LIN {X 0,Y 312.686,Z 295.811,A -85,B 0,C 180,E1 -15649.642,E2 -15649.642} C_VEL
LIN {X 0,Y 312.798,Z 295.834,A -85,B 0,C 180,E1 -15652.253,E2 -15652.253} C_VEL
LIN {X 0,Y 312.699,Z 295.812,A -85,B 0,C 180,E1 -15654.843,E2 -15654.843} C_VEL
LIN {X 0,Y 312.984,Z 295.813,A -85,B 0,C 180,E1 -15658.714,E2 -15658.714} C_VEL
LIN {X 0,Y 312.982,Z 295.778,A -85,B 0,C 180,E1 -15661.287,E2 -15661.287} C_VEL
LIN {X 0,Y 312.841,Z 295.81,A -85,B 0,C 180,E1 -15666.484,E2 -15666.484} C_VEL
LIN {X 0,Y 312.753,Z 295.811,A -85,B 0,C 180,E1 -15669.051,E2 -15669.051} C_VEL
LIN {X 0,Y 312.634,Z 295.828,A -85,B 0,C 180,E1 -15672.992,E2 -15672.992} C_VEL
LIN {X 0,Y 312.615,Z 295.845,A -85,B 0,C 180,E1 -15675.652,E2 -15675.652} C_VEL
LIN {X 0,Y 312.536,Z 295.84,A -85,B 0,C 180,E1 -15679.714,E2 -15679.714} C_VEL
LIN {X 0,Y 312.516,Z 295.853,A -85,B 0,C 180,E1 -15682.775,E2 -15682.775} C_VEL
LIN {X 0,Y 312.491,Z 295.872,A -85,B 0,C 180,E1 -15684.987,E2 -15684.987} C_VEL
LIN {X 0,Y 313.356,Z 298.462,A -85,B 0,C 180,E1 -15685.341,E2 -15685.341} C_VEL
LIN {X 0,Y 315.346,Z 300.712,A -85,B 0,C 180,E1 -15685.986,E2 -15685.986} C_VEL
LIN {X 0,Y 316.693,Z 301.792,A -85,B 0,C 180,E1 -15686.394,E2 -15686.394} C_VEL
LIN {X 0,Y 318.598,Z 304.879,A -85,B 0,C 180,E1 -15687.019,E2 -15687.019} C_VEL
LIN {X 0,Y 320.808,Z 307.144,A -85,B 0,C 180,E1 -15687.673,E2 -15687.673} C_VEL
LIN {X 0,Y 323.371,Z 310.64,A -85,B 0,C 180,E1 -15688.44,E2 -15688.44} C_VEL
LIN {X 0,Y 324.737,Z 312.319,A -85,B 0,C 180,E1 -15688.831,E2 -15688.831} C_VEL
LIN {X 0,Y 328.562,Z 317.398,A -85,B 0,C 180,E1 -15689.896,E2 -15689.896} C_VEL
LIN {X 0,Y 334.896,Z 325.991,A -85,B 0,C 180,E1 -15691.559,E2 -15691.559} C_VEL
LIN {X 0,Y 343.13,Z 338.066,A -85,B 0,C 180,E1 -15693.575,E2 -15693.575} C_VEL
LIN {X 0,Y 348.752,Z 347.569,A -85,B 0,C 180,E1 -15694.885,E2 -15694.885} C_VEL
LIN {X 0,Y 355.328,Z 359.808,A -85,B 0,C 180,E1 -15696.353,E2 -15696.353} C_VEL
LIN {X 0,Y 348.994,Z 496.214,A -85,B 0,C 180,E1 -15699.224,E2 -15699.224} C_VEL
LIN {X 0,Y 347.586,Z 511.917,A -85,B 0,C 180,E1 -15699.738,E2 -15699.738} C_VEL
LIN {X 0,Y 345.628,Z 527.82,A -85,B 0,C 180,E1 -15700.466,E2 -15700.466} C_VEL
LIN {X 0,Y 343.213,Z 543.442,A -85,B 0,C 180,E1 -15701.412,E2 -15701.412} C_VEL
LIN {X 0,Y 340.307,Z 559.032,A -85,B 0,C 180,E1 -15702.615,E2 -15702.615} C_VEL
LIN {X 0,Y 337.092,Z 573.52,A -85,B 0,C 180,E1 -15704.004,E2 -15704.004} C_VEL
LIN {X 0,Y 333.707,Z 587.157,A -85,B 0,C 180,E1 -15705.595,E2 -15705.595} C_VEL
LIN {X 0,Y 330.15,Z 600.476,A -85,B 0,C 180,E1 -15707.478,E2 -15707.478} C_VEL
LIN {X 0,Y 326.807,Z 612.047,A -85,B 0,C 180,E1 -15709.427,E2 -15709.427} C_VEL
LIN {X 0,Y 323.531,Z 622.668,A -85,B 0,C 180,E1 -15711.558,E2 -15711.558} C_VEL
LIN {X 0,Y 320.715,Z 631.72,A -85,B 0,C 180,E1 -15713.724,E2 -15713.724} C_VEL
LIN {X 0,Y 317.842,Z 641.178,A -85,B 0,C 180,E1 -15716.441,E2 -15716.441} C_VEL
LIN {X 0,Y 315.491,Z 648.981,A -85,B 0,C 180,E1 -15719.179,E2 -15719.179} C_VEL
LIN {X 0,Y 313.706,Z 655.293,A -85,B 0,C 180,E1 -15721.935,E2 -15721.935} C_VEL
LIN {X 0,Y 312.36,Z 660.271,A -85,B 0,C 180,E1 -15724.691,E2 -15724.691} C_VEL
LIN {X 0,Y 311.406,Z 664.401,A -85,B 0,C 180,E1 -15727.717,E2 -15727.717} C_VEL
LIN {X 0,Y 310.878,Z 666.76,A -85,B 0,C 180,E1 -15730.178,E2 -15730.178} C_VEL
LIN {X 0,Y 310.594,Z 668.373,A -85,B 0,C 180,E1 -15732.893,E2 -15732.893} C_VEL
LIN {X 0,Y 310.522,Z 668.972,A -85,B 0,C 180,E1 -15735.584,E2 -15735.584} C_VEL
LIN {X 0,Y 310.539,Z 668.546,A -85,B 0,C 180,E1 -15738.247,E2 -15738.247} C_VEL
LIN {X 0,Y 310.551,Z 667.191,A -85,B 0,C 180,E1 -15740.885,E2 -15740.885} C_VEL
LIN {X 0,Y 310.957,Z 664.27,A -85,B 0,C 180,E1 -15743.971,E2 -15743.971} C_VEL
LIN {X 0,Y 311.31,Z 660.413,A -85,B 0,C 180,E1 -15746.764,E2 -15746.764} C_VEL
LIN {X 0,Y 311.935,Z 655.765,A -85,B 0,C 180,E1 -15749.354,E2 -15749.354} C_VEL
LIN {X 0,Y 313.296,Z 648.302,A -85,B 0,C 180,E1 -15752.571,E2 -15752.571} C_VEL
LIN {X 0,Y 314.909,Z 639.877,A -85,B 0,C 180,E1 -15755.443,E2 -15755.443} C_VEL
LIN {X 0,Y 316.998,Z 630.802,A -85,B 0,C 180,E1 -15757.965,E2 -15757.965} C_VEL
LIN {X 0,Y 319.443,Z 620.044,A -85,B 0,C 180,E1 -15760.457,E2 -15760.457} C_VEL
LIN {X 0,Y 321.871,Z 608.968,A -85,B 0,C 180,E1 -15762.612,E2 -15762.612} C_VEL
LIN {X 0,Y 324.394,Z 596.962,A -85,B 0,C 180,E1 -15764.587,E2 -15764.587} C_VEL
LIN {X 0,Y 327.032,Z 583.829,A -85,B 0,C 180,E1 -15766.383,E2 -15766.383} C_VEL
LIN {X 0,Y 329.507,Z 570.928,A -85,B 0,C 180,E1 -15767.854,E2 -15767.854} C_VEL
LIN {X 0,Y 332.094,Z 555.577,A -85,B 0,C 180,E1 -15769.309,E2 -15769.309} C_VEL
LIN {X 0,Y 334.275,Z 540.595,A -85,B 0,C 180,E1 -15770.459,E2 -15770.459} C_VEL
LIN {X 0,Y 335.936,Z 526.536,A -85,B 0,C 180,E1 -15771.315,E2 -15771.315} C_VEL
LIN {X 0,Y 337.496,Z 510.651,A -85,B 0,C 180,E1 -15772.054,E2 -15772.054} C_VEL
LIN {X 0,Y 338.691,Z 494.724,A -85,B 0,C 180,E1 -15772.574,E2 -15772.574} C_VEL
LIN {X 0,Y 341.33,Z 421.868,A -85,B 0,C 180,E1 -15774.13,E2 -15774.13} C_VEL
LIN {X 0,Y 340.959,Z 416.07,A -85,B 0,C 180,E1 -15774.315,E2 -15774.315} C_VEL
LIN {X 0,Y 336.956,Z 397.42,A -85,B 0,C 180,E1 -15775.237,E2 -15775.237} C_VEL
LIN {X 0,Y 336.559,Z 391.625,A -85,B 0,C 180,E1 -15775.431,E2 -15775.431} C_VEL
LIN {X 0,Y 338.038,Z 354.66,A -85,B 0,C 180,E1 -15776.204,E2 -15776.204} C_VEL
LIN {X 0,Y 328.733,Z 335.509,A -85,B 0,C 180,E1 -15777.866,E2 -15777.866} C_VEL
LIN {X 0,Y 318.795,Z 318.498,A -85,B 0,C 180,E1 -15779.685,E2 -15779.685} C_VEL
LIN {X 0,Y 309.969,Z 304.705,A -85,B 0,C 180,E1 -15781.395,E2 -15781.395} C_VEL
LIN {X 0,Y 307.637,Z 301.06,A -85,B 0,C 180,E1 -15781.869,E2 -15781.869} C_VEL
LIN {X 0,Y 305.928,Z 298.586,A -85,B 0,C 180,E1 -15782.217,E2 -15782.217} C_VEL
LIN {X 0,Y 305.465,Z 296.743,A -85,B 0,C 180,E1 -15782.352,E2 -15782.352} C_VEL
LIN {X 0,Y 305.464,Z 296.749,A -85,B 0,C 180,E1 -15786.363,E2 -15786.363} C_VEL
LIN {X 0,Y 305.412,Z 296.756,A -85,B 0,C 180,E1 -15790.115,E2 -15790.115} C_VEL
LIN {X 0,Y 305.422,Z 296.75,A -85,B 0,C 180,E1 -15793.656,E2 -15793.656} C_VEL
LIN {X 0,Y 305.436,Z 296.74,A -85,B 0,C 180,E1 -15797.418,E2 -15797.418} C_VEL
LIN {X 0,Y 305.449,Z 296.709,A -85,B 0,C 180,E1 -15801.593,E2 -15801.593} C_VEL
LIN {X 0,Y 305.462,Z 296.701,A -85,B 0,C 180,E1 -15804.886,E2 -15804.886} C_VEL
LIN {X 0,Y 305.443,Z 296.75,A -85,B 0,C 180,E1 -15808.358,E2 -15808.358} C_VEL
LIN {X 0,Y 305.455,Z 296.731,A -85,B 0,C 180,E1 -15811.106,E2 -15811.106} C_VEL
LIN {X 0,Y 305.499,Z 296.741,A -85,B 0,C 180,E1 -15814.081,E2 -15814.081} C_VEL
LIN {X 0,Y 305.475,Z 296.73,A -85,B 0,C 180,E1 -15816.975,E2 -15816.975} C_VEL
LIN {X 0,Y 305.544,Z 296.724,A -85,B 0,C 180,E1 -15821.214,E2 -15821.214} C_VEL
LIN {X 0,Y 305.628,Z 296.729,A -85,B 0,C 180,E1 -15825.347,E2 -15825.347} C_VEL
LIN {X 0,Y 305.636,Z 296.713,A -85,B 0,C 180,E1 -15829.399,E2 -15829.399} C_VEL
LIN {X 0,Y 305.772,Z 296.706,A -85,B 0,C 180,E1 -15832.073,E2 -15832.073} C_VEL
LIN {X 0,Y 305.675,Z 296.702,A -85,B 0,C 180,E1 -15834.722,E2 -15834.722} C_VEL
LIN {X 0,Y 305.954,Z 296.681,A -85,B 0,C 180,E1 -15838.683,E2 -15838.683} C_VEL
LIN {X 0,Y 305.954,Z 296.669,A -85,B 0,C 180,E1 -15841.316,E2 -15841.316} C_VEL
LIN {X 0,Y 305.679,Z 296.707,A -85,B 0,C 180,E1 -15845.276,E2 -15845.276} C_VEL
LIN {X 0,Y 305.799,Z 296.68,A -85,B 0,C 180,E1 -15847.925,E2 -15847.925} C_VEL
LIN {X 0,Y 305.603,Z 296.725,A -85,B 0,C 180,E1 -15851.944,E2 -15851.944} C_VEL
LIN {X 0,Y 305.608,Z 296.729,A -85,B 0,C 180,E1 -15855.014,E2 -15855.014} C_VEL
LIN {X 0,Y 305.56,Z 296.734,A -85,B 0,C 180,E1 -15859.436,E2 -15859.436} C_VEL
LIN {X 0,Y 305.49,Z 296.744,A -85,B 0,C 180,E1 -15863.041,E2 -15863.041} C_VEL
LIN {X 0,Y 305.53,Z 296.741,A -85,B 0,C 180,E1 -15866.22,E2 -15866.22} C_VEL
LIN {X 0,Y 305.487,Z 296.746,A -85,B 0,C 180,E1 -15869.047,E2 -15869.047} C_VEL
LIN {X 0,Y 305.44,Z 296.752,A -85,B 0,C 180,E1 -15871.952,E2 -15871.952} C_VEL
LIN {X 0,Y 305.461,Z 296.744,A -85,B 0,C 180,E1 -15875.113,E2 -15875.113} C_VEL
LIN {X 0,Y 305.465,Z 296.748,A -85,B 0,C 180,E1 -15878.533,E2 -15878.533} C_VEL
LIN {X 0,Y 305.457,Z 296.753,A -85,B 0,C 180,E1 -15882.586,E2 -15882.586} C_VEL
LIN {X 0,Y 305.427,Z 296.81,A -85,B 0,C 180,E1 -15883.063,E2 -15883.063} C_VEL
LIN {X 0,Y 308.169,Z 304.268,A -85,B 0,C 180,E1 -15884.928,E2 -15884.928} C_VEL
LIN {X 0,Y 316.716,Z 319.019,A -85,B 0,C 180,E1 -15886.646,E2 -15886.646} C_VEL
LIN {X 0,Y 323.706,Z 332.142,A -85,B 0,C 180,E1 -15887.992,E2 -15887.992} C_VEL
LIN {X 0,Y 332.604,Z 350.491,A -85,B 0,C 180,E1 -15889.641,E2 -15889.641} C_VEL
LIN {X 0,Y 337.927,Z 362.483,A -85,B 0,C 180,E1 -15890.598,E2 -15890.598} C_VEL
LIN {X 0,Y 332.319,Z 511.428,A -85,B 0,C 180,E1 -15893.784,E2 -15893.784} C_VEL
LIN {X 0,Y 331.012,Z 527.703,A -85,B 0,C 180,E1 -15894.323,E2 -15894.323} C_VEL
LIN {X 0,Y 329.18,Z 543.894,A -85,B 0,C 180,E1 -15895.079,E2 -15895.079} C_VEL
LIN {X 0,Y 327.159,Z 559.351,A -85,B 0,C 180,E1 -15896.046,E2 -15896.046} C_VEL
LIN {X 0,Y 324.616,Z 574.513,A -85,B 0,C 180,E1 -15897.231,E2 -15897.231} C_VEL
LIN {X 0,Y 322.08,Z 588.525,A -85,B 0,C 180,E1 -15898.603,E2 -15898.603} C_VEL
LIN {X 0,Y 319.117,Z 602.903,A -85,B 0,C 180,E1 -15900.296,E2 -15900.296} C_VEL
LIN {X 0,Y 316.291,Z 616.145,A -85,B 0,C 180,E1 -15902.185,E2 -15902.185} C_VEL
LIN {X 0,Y 313.742,Z 627.491,A -85,B 0,C 180,E1 -15904.1,E2 -15904.1} C_VEL
LIN {X 0,Y 311.182,Z 638.736,A -85,B 0,C 180,E1 -15906.367,E2 -15906.367} C_VEL
LIN {X 0,Y 309.055,Z 648.356,A -85,B 0,C 180,E1 -15908.664,E2 -15908.664} C_VEL
LIN {X 0,Y 307.152,Z 657.693,A -85,B 0,C 180,E1 -15911.317,E2 -15911.317} C_VEL
LIN {X 0,Y 305.648,Z 665.471,A -85,B 0,C 180,E1 -15913.983,E2 -15913.983} C_VEL
LIN {X 0,Y 304.665,Z 671.817,A -85,B 0,C 180,E1 -15916.663,E2 -15916.663} C_VEL
LIN {X 0,Y 303.958,Z 676.988,A -85,B 0,C 180,E1 -15919.341,E2 -15919.341} C_VEL
LIN {X 0,Y 303.682,Z 680.998,A -85,B 0,C 180,E1 -15922.019,E2 -15922.019} C_VEL
LIN {X 0,Y 303.614,Z 683.933,A -85,B 0,C 180,E1 -15924.687,E2 -15924.687} C_VEL
LIN {X 0,Y 303.601,Z 685.852,A -85,B 0,C 180,E1 -15927.347,E2 -15927.347} C_VEL
LIN {X 0,Y 303.602,Z 686.754,A -85,B 0,C 180,E1 -15930,E2 -15930} C_VEL
LIN {X 0,Y 303.592,Z 686.701,A -85,B 0,C 180,E1 -15932.654,E2 -15932.654} C_VEL
LIN {X 0,Y 303.621,Z 685.522,A -85,B 0,C 180,E1 -15935.545,E2 -15935.545} C_VEL
LIN {X 0,Y 303.688,Z 683.676,A -85,B 0,C 180,E1 -15937.982,E2 -15937.982} C_VEL
LIN {X 0,Y 304.027,Z 680.69,A -85,B 0,C 180,E1 -15940.657,E2 -15940.657} C_VEL
LIN {X 0,Y 304.827,Z 676.704,A -85,B 0,C 180,E1 -15943.33,E2 -15943.33} C_VEL
LIN {X 0,Y 305.923,Z 671.604,A -85,B 0,C 180,E1 -15946.003,E2 -15946.003} C_VEL
LIN {X 0,Y 307.626,Z 665.419,A -85,B 0,C 180,E1 -15948.654,E2 -15948.654} C_VEL
LIN {X 0,Y 309.772,Z 657.865,A -85,B 0,C 180,E1 -15951.285,E2 -15951.285} C_VEL
LIN {X 0,Y 312.559,Z 648.91,A -85,B 0,C 180,E1 -15953.875,E2 -15953.875} C_VEL
LIN {X 0,Y 315.874,Z 638.315,A -85,B 0,C 180,E1 -15956.423,E2 -15956.423} C_VEL
LIN {X 0,Y 319.215,Z 627.6,A -85,B 0,C 180,E1 -15958.575,E2 -15958.575} C_VEL
LIN {X 0,Y 322.531,Z 616.502,A -85,B 0,C 180,E1 -15960.439,E2 -15960.439} C_VEL
LIN {X 0,Y 325.907,Z 605.036,A -85,B 0,C 180,E1 -15962.075,E2 -15962.075} C_VEL
LIN {X 0,Y 329.415,Z 591.636,A -85,B 0,C 180,E1 -15963.691,E2 -15963.691} C_VEL
LIN {X 0,Y 332.99,Z 577.061,A -85,B 0,C 180,E1 -15965.109,E2 -15965.109} C_VEL
LIN {X 0,Y 335.929,Z 563.101,A -85,B 0,C 180,E1 -15966.23,E2 -15966.23} C_VEL
LIN {X 0,Y 338.617,Z 548.294,A -85,B 0,C 180,E1 -15967.192,E2 -15967.192} C_VEL
LIN {X 0,Y 341.085,Z 531.799,A -85,B 0,C 180,E1 -15967.994,E2 -15967.994} C_VEL
LIN {X 0,Y 342.849,Z 515.977,A -85,B 0,C 180,E1 -15968.542,E2 -15968.542} C_VEL
LIN {X 0,Y 344.097,Z 495.089,A -85,B 0,C 180,E1 -15969.047,E2 -15969.047} C_VEL
LIN {X 0,Y 349.94,Z 369.642,A -85,B 0,C 180,E1 -15971.705,E2 -15971.705} C_VEL
LIN {X 0,Y 342.001,Z 354.097,A -85,B 0,C 180,E1 -15973.584,E2 -15973.584} C_VEL
LIN {X 0,Y 334.526,Z 340.991,A -85,B 0,C 180,E1 -15975.465,E2 -15975.465} C_VEL
LIN {X 0,Y 327.373,Z 329.638,A -85,B 0,C 180,E1 -15977.385,E2 -15977.385} C_VEL
LIN {X 0,Y 320.557,Z 319.554,A -85,B 0,C 180,E1 -15979.362,E2 -15979.362} C_VEL
LIN {X 0,Y 316.114,Z 313.396,A -85,B 0,C 180,E1 -15980.742,E2 -15980.742} C_VEL
LIN {X 0,Y 309.814,Z 305.018,A -85,B 0,C 180,E1 -15982.846,E2 -15982.846} C_VEL
LIN {X 0,Y 307.631,Z 301.915,A -85,B 0,C 180,E1 -15983.669,E2 -15983.669} C_VEL
LIN {X 0,Y 305.507,Z 297.046,A -85,B 0,C 180,E1 -15985.756,E2 -15985.756} C_VEL
LIN {X 0,Y 305.464,Z 296.728,A -85,B 0,C 180,E1 -15985.922,E2 -15985.922} C_VEL
LIN {X 0,Y 305.459,Z 296.748,A -85,B 0,C 180,E1 -15989.591,E2 -15989.591} C_VEL
LIN {X 0,Y 305.518,Z 296.713,A -85,B 0,C 180,E1 -15992.609,E2 -15992.609} C_VEL
LIN {X 0,Y 305.505,Z 296.728,A -85,B 0,C 180,E1 -15995.539,E2 -15995.539} C_VEL
LIN {X 0,Y 305.513,Z 296.741,A -85,B 0,C 180,E1 -15999.815,E2 -15999.815} C_VEL
LIN {X 0,Y 305.575,Z 296.7,A -85,B 0,C 180,E1 -16002.604,E2 -16002.604} C_VEL
LIN {X 0,Y 305.65,Z 296.715,A -85,B 0,C 180,E1 -16005.35,E2 -16005.35} C_VEL
LIN {X 0,Y 305.625,Z 296.689,A -85,B 0,C 180,E1 -16009.4,E2 -16009.4} C_VEL
LIN {X 0,Y 305.748,Z 296.711,A -85,B 0,C 180,E1 -16012.073,E2 -16012.073} C_VEL
LIN {X 0,Y 305.668,Z 296.688,A -85,B 0,C 180,E1 -16014.724,E2 -16014.724} C_VEL
LIN {X 0,Y 305.951,Z 296.689,A -85,B 0,C 180,E1 -16018.684,E2 -16018.684} C_VEL
LIN {X 0,Y 305.949,Z 296.653,A -85,B 0,C 180,E1 -16021.317,E2 -16021.317} C_VEL
LIN {X 0,Y 305.789,Z 296.685,A -85,B 0,C 180,E1 -16026.6,E2 -16026.6} C_VEL
LIN {X 0,Y 305.696,Z 296.692,A -85,B 0,C 180,E1 -16029.262,E2 -16029.262} C_VEL
LIN {X 0,Y 305.587,Z 296.702,A -85,B 0,C 180,E1 -16033.297,E2 -16033.297} C_VEL
LIN {X 0,Y 305.543,Z 296.733,A -85,B 0,C 180,E1 -16036.024,E2 -16036.024} C_VEL
LIN {X 0,Y 305.482,Z 296.723,A -85,B 0,C 180,E1 -16040.188,E2 -16040.188} C_VEL
LIN {X 0,Y 305.47,Z 296.729,A -85,B 0,C 180,E1 -16042.879,E2 -16042.879} C_VEL
LIN {X 0,Y 306.272,Z 299.3,A -85,B 0,C 180,E1 -16043.267,E2 -16043.267} C_VEL
LIN {X 0,Y 308.202,Z 301.528,A -85,B 0,C 180,E1 -16043.966,E2 -16043.966} C_VEL
LIN {X 0,Y 309.717,Z 302.518,A -85,B 0,C 180,E1 -16044.465,E2 -16044.465} C_VEL
LIN {X 0,Y 311.507,Z 305.592,A -85,B 0,C 180,E1 -16045.116,E2 -16045.116} C_VEL
LIN {X 0,Y 313.981,Z 308.059,A -85,B 0,C 180,E1 -16045.912,E2 -16045.912} C_VEL
LIN {X 0,Y 316.359,Z 311.432,A -85,B 0,C 180,E1 -16046.691,E2 -16046.691} C_VEL
LIN {X 0,Y 317.908,Z 313.042,A -85,B 0,C 180,E1 -16047.161,E2 -16047.161} C_VEL
LIN {X 0,Y 320.945,Z 317.023,A -85,B 0,C 180,E1 -16048.085,E2 -16048.085} C_VEL
LIN {X 0,Y 325.541,Z 323.245,A -85,B 0,C 180,E1 -16049.417,E2 -16049.417} C_VEL
LIN {X 0,Y 332.025,Z 332.219,A -85,B 0,C 180,E1 -16051.166,E2 -16051.166} C_VEL
LIN {X 0,Y 339.376,Z 343.096,A -85,B 0,C 180,E1 -16053.018,E2 -16053.018} C_VEL
LIN {X 0,Y 344.768,Z 352.352,A -85,B 0,C 180,E1 -16054.317,E2 -16054.317} C_VEL
LIN {X 0,Y 350.248,Z 362.537,A -85,B 0,C 180,E1 -16055.586,E2 -16055.586} C_VEL
LIN {X 0,Y 343.759,Z 496.864,A -85,B 0,C 180,E1 -16058.442,E2 -16058.442} C_VEL
LIN {X 0,Y 342.305,Z 512.312,A -85,B 0,C 180,E1 -16058.956,E2 -16058.956} C_VEL
LIN {X 0,Y 340.414,Z 527.383,A -85,B 0,C 180,E1 -16059.651,E2 -16059.651} C_VEL
LIN {X 0,Y 337.874,Z 543.192,A -85,B 0,C 180,E1 -16060.604,E2 -16060.604} C_VEL
LIN {X 0,Y 334.822,Z 558.968,A -85,B 0,C 180,E1 -16061.828,E2 -16061.828} C_VEL
LIN {X 0,Y 331.523,Z 573.382,A -85,B 0,C 180,E1 -16063.22,E2 -16063.22} C_VEL
LIN {X 0,Y 328.055,Z 586.826,A -85,B 0,C 180,E1 -16064.794,E2 -16064.794} C_VEL
LIN {X 0,Y 324.267,Z 600.442,A -85,B 0,C 180,E1 -16066.731,E2 -16066.731} C_VEL
LIN {X 0,Y 320.961,Z 611.512,A -85,B 0,C 180,E1 -16068.605,E2 -16068.605} C_VEL
LIN {X 0,Y 317.441,Z 622.344,A -85,B 0,C 180,E1 -16070.796,E2 -16070.796} C_VEL
LIN {X 0,Y 314.234,Z 632.134,A -85,B 0,C 180,E1 -16073.169,E2 -16073.169} C_VEL
LIN {X 0,Y 311.495,Z 640.718,A -85,B 0,C 180,E1 -16075.663,E2 -16075.663} C_VEL
LIN {X 0,Y 308.963,Z 648.648,A -85,B 0,C 180,E1 -16078.454,E2 -16078.454} C_VEL
LIN {X 0,Y 307.008,Z 655.035,A -85,B 0,C 180,E1 -16081.267,E2 -16081.267} C_VEL
LIN {X 0,Y 305.53,Z 660.135,A -85,B 0,C 180,E1 -16084.084,E2 -16084.084} C_VEL
LIN {X 0,Y 304.548,Z 664.073,A -85,B 0,C 180,E1 -16086.902,E2 -16086.902} C_VEL
LIN {X 0,Y 303.888,Z 666.788,A -85,B 0,C 180,E1 -16089.702,E2 -16089.702} C_VEL
LIN {X 0,Y 303.537,Z 668.506,A -85,B 0,C 180,E1 -16092.482,E2 -16092.482} C_VEL
LIN {X 0,Y 303.42,Z 669.157,A -85,B 0,C 180,E1 -16095.239,E2 -16095.239} C_VEL
LIN {X 0,Y 303.433,Z 668.835,A -85,B 0,C 180,E1 -16097.968,E2 -16097.968} C_VEL
LIN {X 0,Y 303.445,Z 667.529,A -85,B 0,C 180,E1 -16100.67,E2 -16100.67} C_VEL
LIN {X 0,Y 303.883,Z 664.542,A -85,B 0,C 180,E1 -16103.983,E2 -16103.983} C_VEL
LIN {X 0,Y 304.194,Z 660.962,A -85,B 0,C 180,E1 -16106.689,E2 -16106.689} C_VEL
LIN {X 0,Y 304.852,Z 656.366,A -85,B 0,C 180,E1 -16109.339,E2 -16109.339} C_VEL
LIN {X 0,Y 305.899,Z 650.613,A -85,B 0,C 180,E1 -16111.975,E2 -16111.975} C_VEL
LIN {X 0,Y 307.221,Z 643.701,A -85,B 0,C 180,E1 -16114.592,E2 -16114.592} C_VEL
LIN {X 0,Y 309.122,Z 635.333,A -85,B 0,C 180,E1 -16117.183,E2 -16117.183} C_VEL
LIN {X 0,Y 311.52,Z 625.363,A -85,B 0,C 180,E1 -16119.741,E2 -16119.741} C_VEL
LIN {X 0,Y 313.901,Z 615.131,A -85,B 0,C 180,E1 -16121.952,E2 -16121.952} C_VEL
LIN {X 0,Y 316.599,Z 603.168,A -85,B 0,C 180,E1 -16124.133,E2 -16124.133} C_VEL
LIN {X 0,Y 319.2,Z 591.124,A -85,B 0,C 180,E1 -16125.975,E2 -16125.975} C_VEL
LIN {X 0,Y 321.797,Z 578.151,A -85,B 0,C 180,E1 -16127.639,E2 -16127.639} C_VEL
LIN {X 0,Y 324.447,Z 564.219,A -85,B 0,C 180,E1 -16129.125,E2 -16129.125} C_VEL
LIN {X 0,Y 326.846,Z 549.19,A -85,B 0,C 180,E1 -16130.451,E2 -16130.451} C_VEL
LIN {X 0,Y 328.957,Z 533.645,A -85,B 0,C 180,E1 -16131.543,E2 -16131.543} C_VEL
LIN {X 0,Y 330.945,Z 516.706,A -85,B 0,C 180,E1 -16132.432,E2 -16132.432} C_VEL
LIN {X 0,Y 332.211,Z 501.941,A -85,B 0,C 180,E1 -16132.999,E2 -16132.999} C_VEL
LIN {X 0,Y 333.161,Z 484.122,A -85,B 0,C 180,E1 -16133.463,E2 -16133.463} C_VEL
LIN {X 0,Y 336.559,Z 391.625,A -85,B 0,C 180,E1 -16135.431,E2 -16135.431} C_VEL
LIN {X 0,Y 336.151,Z 385.828,A -85,B 0,C 180,E1 -16135.627,E2 -16135.627} C_VEL
LIN {X 0,Y 332.238,Z 367.184,A -85,B 0,C 180,E1 -16136.581,E2 -16136.581} C_VEL
LIN {X 0,Y 331.992,Z 361.383,A -85,B 0,C 180,E1 -16136.764,E2 -16136.764} C_VEL
LIN {X 0,Y 332.117,Z 356.706,A -85,B 0,C 180,E1 -16136.872,E2 -16136.872} C_VEL
LIN {X 0,Y 323.631,Z 339.316,A -85,B 0,C 180,E1 -16138.434,E2 -16138.434} C_VEL
LIN {X 0,Y 314.098,Z 322.876,A -85,B 0,C 180,E1 -16140.239,E2 -16140.239} C_VEL
LIN {X 0,Y 305.424,Z 309.288,A -85,B 0,C 180,E1 -16141.97,E2 -16141.97} C_VEL
LIN {X 0,Y 303.104,Z 305.75,A -85,B 0,C 180,E1 -16142.455,E2 -16142.455} C_VEL
LIN {X 0,Y 300.673,Z 301.985,A -85,B 0,C 180,E1 -16142.976,E2 -16142.976} C_VEL
LIN {X 0,Y 298.963,Z 299.557,A -85,B 0,C 180,E1 -16143.344,E2 -16143.344} C_VEL
LIN {X 0,Y 298.436,Z 297.626,A -85,B 0,C 180,E1 -16143.515,E2 -16143.515} C_VEL
LIN {X 0,Y 298.389,Z 297.62,A -85,B 0,C 180,E1 -16147.762,E2 -16147.762} C_VEL
LIN {X 0,Y 298.349,Z 297.625,A -85,B 0,C 180,E1 -16151.267,E2 -16151.267} C_VEL
LIN {X 0,Y 298.357,Z 297.629,A -85,B 0,C 180,E1 -16155.034,E2 -16155.034} C_VEL
LIN {X 0,Y 298.349,Z 297.634,A -85,B 0,C 180,E1 -16158.921,E2 -16158.921} C_VEL
LIN {X 0,Y 298.427,Z 297.564,A -85,B 0,C 180,E1 -16163.197,E2 -16163.197} C_VEL
LIN {X 0,Y 298.394,Z 297.623,A -85,B 0,C 180,E1 -16167.199,E2 -16167.199} C_VEL
LIN {X 0,Y 298.366,Z 297.613,A -85,B 0,C 180,E1 -16170.637,E2 -16170.637} C_VEL
LIN {X 0,Y 298.439,Z 297.615,A -85,B 0,C 180,E1 -16174.919,E2 -16174.919} C_VEL
LIN {X 0,Y 298.404,Z 297.619,A -85,B 0,C 180,E1 -16177.862,E2 -16177.862} C_VEL
LIN {X 0,Y 298.505,Z 297.606,A -85,B 0,C 180,E1 -16180.754,E2 -16180.754} C_VEL
LIN {X 0,Y 298.587,Z 297.604,A -85,B 0,C 180,E1 -16184.994,E2 -16184.994} C_VEL
LIN {X 0,Y 298.592,Z 297.588,A -85,B 0,C 180,E1 -16189.146,E2 -16189.146} C_VEL
LIN {X 0,Y 298.718,Z 297.585,A -85,B 0,C 180,E1 -16191.884,E2 -16191.884} C_VEL
LIN {X 0,Y 298.645,Z 297.576,A -85,B 0,C 180,E1 -16194.598,E2 -16194.598} C_VEL
LIN {X 0,Y 298.92,Z 297.557,A -85,B 0,C 180,E1 -16198.652,E2 -16198.652} C_VEL
LIN {X 0,Y 298.921,Z 297.545,A -85,B 0,C 180,E1 -16201.346,E2 -16201.346} C_VEL
LIN {X 0,Y 298.65,Z 297.58,A -85,B 0,C 180,E1 -16205.401,E2 -16205.401} C_VEL
LIN {X 0,Y 298.743,Z 297.56,A -85,B 0,C 180,E1 -16208.114,E2 -16208.114} C_VEL
LIN {X 0,Y 298.553,Z 297.602,A -85,B 0,C 180,E1 -16212.231,E2 -16212.231} C_VEL
LIN {X 0,Y 298.548,Z 297.607,A -85,B 0,C 180,E1 -16215.168,E2 -16215.168} C_VEL
LIN {X 0,Y 298.52,Z 297.61,A -85,B 0,C 180,E1 -16219.244,E2 -16219.244} C_VEL
LIN {X 0,Y 298.457,Z 297.624,A -85,B 0,C 180,E1 -16223.597,E2 -16223.597} C_VEL
LIN {X 0,Y 298.485,Z 297.62,A -85,B 0,C 180,E1 -16226.574,E2 -16226.574} C_VEL
LIN {X 0,Y 298.415,Z 297.628,A -85,B 0,C 180,E1 -16229.641,E2 -16229.641} C_VEL
LIN {X 0,Y 298.393,Z 297.627,A -85,B 0,C 180,E1 -16232.8,E2 -16232.8} C_VEL
LIN {X 0,Y 298.445,Z 297.605,A -85,B 0,C 180,E1 -16236.807,E2 -16236.807} C_VEL
LIN {X 0,Y 298.407,Z 297.624,A -85,B 0,C 180,E1 -16239.486,E2 -16239.486} C_VEL
LIN {X 0,Y 298.431,Z 297.817,A -85,B 0,C 180,E1 -16242.1,E2 -16242.1} C_VEL
LIN {X 0,Y 300.758,Z 303.975,A -85,B 0,C 180,E1 -16243.716,E2 -16243.716} C_VEL
LIN {X 0,Y 310.516,Z 320.667,A -85,B 0,C 180,E1 -16245.78,E2 -16245.78} C_VEL
LIN {X 0,Y 318.198,Z 335.006,A -85,B 0,C 180,E1 -16247.313,E2 -16247.313} C_VEL
LIN {X 0,Y 327.233,Z 353.65,A -85,B 0,C 180,E1 -16249.044,E2 -16249.044} C_VEL
LIN {X 0,Y 332.038,Z 364.587,A -85,B 0,C 180,E1 -16249.942,E2 -16249.942} C_VEL
LIN {X 0,Y 326.268,Z 512.099,A -85,B 0,C 180,E1 -16253.147,E2 -16253.147} C_VEL
LIN {X 0,Y 324.827,Z 528.962,A -85,B 0,C 180,E1 -16253.729,E2 -16253.729} C_VEL
LIN {X 0,Y 322.946,Z 544.74,A -85,B 0,C 180,E1 -16254.495,E2 -16254.495} C_VEL
LIN {X 0,Y 320.713,Z 560.972,A -85,B 0,C 180,E1 -16255.553,E2 -16255.553} C_VEL
LIN {X 0,Y 317.909,Z 576.606,A -85,B 0,C 180,E1 -16256.826,E2 -16256.826} C_VEL
LIN {X 0,Y 315.073,Z 591.772,A -85,B 0,C 180,E1 -16258.386,E2 -16258.386} C_VEL
LIN {X 0,Y 312.083,Z 605.599,A -85,B 0,C 180,E1 -16260.116,E2 -16260.116} C_VEL
LIN {X 0,Y 309.424,Z 617.357,A -85,B 0,C 180,E1 -16261.882,E2 -16261.882} C_VEL
LIN {X 0,Y 306.841,Z 628.501,A -85,B 0,C 180,E1 -16263.838,E2 -16263.838} C_VEL
LIN {X 0,Y 304.201,Z 639.609,A -85,B 0,C 180,E1 -16266.153,E2 -16266.153} C_VEL
LIN {X 0,Y 301.939,Z 649.407,A -85,B 0,C 180,E1 -16268.597,E2 -16268.597} C_VEL
LIN {X 0,Y 300.067,Z 658.219,A -85,B 0,C 180,E1 -16271.214,E2 -16271.214} C_VEL
LIN {X 0,Y 298.712,Z 664.999,A -85,B 0,C 180,E1 -16273.601,E2 -16273.601} C_VEL
LIN {X 0,Y 297.676,Z 671.406,A -85,B 0,C 180,E1 -16276.344,E2 -16276.344} C_VEL
LIN {X 0,Y 296.908,Z 676.63,A -85,B 0,C 180,E1 -16279.084,E2 -16279.084} C_VEL
LIN {X 0,Y 296.614,Z 680.667,A -85,B 0,C 180,E1 -16281.827,E2 -16281.827} C_VEL
LIN {X 0,Y 296.548,Z 683.65,A -85,B 0,C 180,E1 -16284.56,E2 -16284.56} C_VEL
LIN {X 0,Y 296.526,Z 685.591,A -85,B 0,C 180,E1 -16287.283,E2 -16287.283} C_VEL
LIN {X 0,Y 296.517,Z 686.535,A -85,B 0,C 180,E1 -16290,E2 -16290} C_VEL
LIN {X 0,Y 296.516,Z 686.505,A -85,B 0,C 180,E1 -16292.717,E2 -16292.717} C_VEL
LIN {X 0,Y 296.508,Z 685.511,A -85,B 0,C 180,E1 -16295.441,E2 -16295.441} C_VEL
LIN {X 0,Y 296.621,Z 683.546,A -85,B 0,C 180,E1 -16298.173,E2 -16298.173} C_VEL
LIN {X 0,Y 296.986,Z 680.606,A -85,B 0,C 180,E1 -16300.913,E2 -16300.913} C_VEL
LIN {X 0,Y 297.848,Z 676.644,A -85,B 0,C 180,E1 -16303.648,E2 -16303.648} C_VEL
LIN {X 0,Y 299.012,Z 671.596,A -85,B 0,C 180,E1 -16306.383,E2 -16306.383} C_VEL
LIN {X 0,Y 300.828,Z 665.443,A -85,B 0,C 180,E1 -16309.091,E2 -16309.091} C_VEL
LIN {X 0,Y 303.468,Z 656.884,A -85,B 0,C 180,E1 -16312.128,E2 -16312.128} C_VEL
LIN {X 0,Y 306.416,Z 647.843,A -85,B 0,C 180,E1 -16314.745,E2 -16314.745} C_VEL
LIN {X 0,Y 309.971,Z 637.143,A -85,B 0,C 180,E1 -16317.314,E2 -16317.314} C_VEL
LIN {X 0,Y 313.567,Z 626.004,A -85,B 0,C 180,E1 -16319.544,E2 -16319.544} C_VEL
LIN {X 0,Y 317.591,Z 612.979,A -85,B 0,C 180,E1 -16321.707,E2 -16321.707} C_VEL
LIN {X 0,Y 321.838,Z 598.764,A -85,B 0,C 180,E1 -16323.618,E2 -16323.618} C_VEL
LIN {X 0,Y 325.389,Z 585.329,A -85,B 0,C 180,E1 -16325.105,E2 -16325.105} C_VEL
LIN {X 0,Y 328.768,Z 571.267,A -85,B 0,C 180,E1 -16326.385,E2 -16326.385} C_VEL
LIN {X 0,Y 331.9,Z 556.173,A -85,B 0,C 180,E1 -16327.502,E2 -16327.502} C_VEL
LIN {X 0,Y 334.298,Z 542.026,A -85,B 0,C 180,E1 -16328.33,E2 -16328.33} C_VEL
LIN {X 0,Y 336.603,Z 525.612,A -85,B 0,C 180,E1 -16329.045,E2 -16329.045} C_VEL
LIN {X 0,Y 338.277,Z 508.622,A -85,B 0,C 180,E1 -16329.557,E2 -16329.557} C_VEL
LIN {X 0,Y 344.913,Z 372.333,A -85,B 0,C 180,E1 -16332.496,E2 -16332.496} C_VEL
LIN {X 0,Y 337.445,Z 357.745,A -85,B 0,C 180,E1 -16334.335,E2 -16334.335} C_VEL
LIN {X 0,Y 331.112,Z 346.439,A -85,B 0,C 180,E1 -16335.992,E2 -16335.992} C_VEL
LIN {X 0,Y 324.191,Z 335.26,A -85,B 0,C 180,E1 -16337.908,E2 -16337.908} C_VEL
LIN {X 0,Y 317.066,Z 324.592,A -85,B 0,C 180,E1 -16340.051,E2 -16340.051} C_VEL
LIN {X 0,Y 313.067,Z 318.986,A -85,B 0,C 180,E1 -16341.337,E2 -16341.337} C_VEL
LIN {X 0,Y 307.372,Z 311.224,A -85,B 0,C 180,E1 -16343.302,E2 -16343.302} C_VEL
LIN {X 0,Y 303.646,Z 306.318,A -85,B 0,C 180,E1 -16344.697,E2 -16344.697} C_VEL
LIN {X 0,Y 301.002,Z 302.932,A -85,B 0,C 180,E1 -16345.741,E2 -16345.741} C_VEL
LIN {X 0,Y 300.205,Z 301.46,A -85,B 0,C 180,E1 -16346.12,E2 -16346.12} C_VEL
LIN {X 0,Y 298.84,Z 299.363,A -85,B 0,C 180,E1 -16347.256,E2 -16347.256} C_VEL
LIN {X 0,Y 298.397,Z 297.608,A -85,B 0,C 180,E1 -16348.103,E2 -16348.103} C_VEL
LIN {X 0,Y 298.459,Z 297.589,A -85,B 0,C 180,E1 -16351.905,E2 -16351.905} C_VEL
LIN {X 0,Y 298.484,Z 297.615,A -85,B 0,C 180,E1 -16354.925,E2 -16354.925} C_VEL
LIN {X 0,Y 298.441,Z 297.61,A -85,B 0,C 180,E1 -16359.315,E2 -16359.315} C_VEL
LIN {X 0,Y 298.538,Z 297.58,A -85,B 0,C 180,E1 -16362.18,E2 -16362.18} C_VEL
LIN {X 0,Y 298.594,Z 297.585,A -85,B 0,C 180,E1 -16364.996,E2 -16364.996} C_VEL
LIN {X 0,Y 298.584,Z 297.566,A -85,B 0,C 180,E1 -16369.147,E2 -16369.147} C_VEL
LIN {X 0,Y 298.7,Z 297.586,A -85,B 0,C 180,E1 -16371.885,E2 -16371.885} C_VEL
LIN {X 0,Y 298.637,Z 297.565,A -85,B 0,C 180,E1 -16374.599,E2 -16374.599} C_VEL
LIN {X 0,Y 298.918,Z 297.564,A -85,B 0,C 180,E1 -16378.653,E2 -16378.653} C_VEL
LIN {X 0,Y 298.915,Z 297.527,A -85,B 0,C 180,E1 -16381.348,E2 -16381.348} C_VEL
LIN {X 0,Y 298.738,Z 297.56,A -85,B 0,C 180,E1 -16386.756,E2 -16386.756} C_VEL
LIN {X 0,Y 298.627,Z 297.574,A -85,B 0,C 180,E1 -16389.483,E2 -16389.483} C_VEL
LIN {X 0,Y 298.545,Z 297.577,A -85,B 0,C 180,E1 -16393.616,E2 -16393.616} C_VEL
LIN {X 0,Y 298.475,Z 297.619,A -85,B 0,C 180,E1 -16396.414,E2 -16396.414} C_VEL
LIN {X 0,Y 298.419,Z 297.63,A -85,B 0,C 180,E1 -16400.532,E2 -16400.532} C_VEL
LIN {X 0,Y 299.216,Z 300.136,A -85,B 0,C 180,E1 -16400.945,E2 -16400.945} C_VEL
LIN {X 0,Y 300.989,Z 302.254,A -85,B 0,C 180,E1 -16401.668,E2 -16401.668} C_VEL
LIN {X 0,Y 302.861,Z 303.514,A -85,B 0,C 180,E1 -16402.359,E2 -16402.359} C_VEL
LIN {X 0,Y 304.658,Z 306.631,A -85,B 0,C 180,E1 -16403.09,E2 -16403.09} C_VEL
LIN {X 0,Y 307.297,Z 309.146,A -85,B 0,C 180,E1 -16404.028,E2 -16404.028} C_VEL
LIN {X 0,Y 309.809,Z 312.648,A -85,B 0,C 180,E1 -16404.927,E2 -16404.927} C_VEL
LIN {X 0,Y 311.45,Z 314.401,A -85,B 0,C 180,E1 -16405.47,E2 -16405.47} C_VEL
LIN {X 0,Y 314.327,Z 318.14,A -85,B 0,C 180,E1 -16406.417,E2 -16406.417} C_VEL
LIN {X 0,Y 319.247,Z 324.606,A -85,B 0,C 180,E1 -16407.95,E2 -16407.95} C_VEL
LIN {X 0,Y 325.538,Z 333.182,A -85,B 0,C 180,E1 -16409.773,E2 -16409.773} C_VEL
LIN {X 0,Y 333.458,Z 344.711,A -85,B 0,C 180,E1 -16411.886,E2 -16411.886} C_VEL
LIN {X 0,Y 338.995,Z 353.7,A -85,B 0,C 180,E1 -16413.282,E2 -16413.282} C_VEL
LIN {X 0,Y 345.22,Z 365.456,A -85,B 0,C 180,E1 -16414.797,E2 -16414.797} C_VEL
LIN {X 0,Y 338.633,Z 496.889,A -85,B 0,C 180,E1 -16417.62,E2 -16417.62} C_VEL
LIN {X 0,Y 337.082,Z 512.722,A -85,B 0,C 180,E1 -16418.148,E2 -16418.148} C_VEL
LIN {X 0,Y 335.094,Z 528.009,A -85,B 0,C 180,E1 -16418.864,E2 -16418.864} C_VEL
LIN {X 0,Y 332.511,Z 543.514,A -85,B 0,C 180,E1 -16419.81,E2 -16419.81} C_VEL
LIN {X 0,Y 329.457,Z 558.806,A -85,B 0,C 180,E1 -16421.007,E2 -16421.007} C_VEL
LIN {X 0,Y 325.912,Z 573.694,A -85,B 0,C 180,E1 -16422.454,E2 -16422.454} C_VEL
LIN {X 0,Y 322.397,Z 586.757,A -85,B 0,C 180,E1 -16423.997,E2 -16423.997} C_VEL
LIN {X 0,Y 318.793,Z 599.387,A -85,B 0,C 180,E1 -16425.798,E2 -16425.798} C_VEL
LIN {X 0,Y 314.809,Z 612.022,A -85,B 0,C 180,E1 -16427.953,E2 -16427.953} C_VEL
LIN {X 0,Y 310.911,Z 623.576,A -85,B 0,C 180,E1 -16430.345,E2 -16430.345} C_VEL
LIN {X 0,Y 307.633,Z 633.073,A -85,B 0,C 180,E1 -16432.732,E2 -16432.732} C_VEL
LIN {X 0,Y 304.466,Z 642.377,A -85,B 0,C 180,E1 -16435.56,E2 -16435.56} C_VEL
LIN {X 0,Y 301.876,Z 650.016,A -85,B 0,C 180,E1 -16438.411,E2 -16438.411} C_VEL
LIN {X 0,Y 299.902,Z 656.247,A -85,B 0,C 180,E1 -16441.288,E2 -16441.288} C_VEL
LIN {X 0,Y 298.109,Z 662.166,A -85,B 0,C 180,E1 -16444.89,E2 -16444.89} C_VEL
LIN {X 0,Y 297.221,Z 665.539,A -85,B 0,C 180,E1 -16447.769,E2 -16447.769} C_VEL
LIN {X 0,Y 296.666,Z 667.852,A -85,B 0,C 180,E1 -16450.63,E2 -16450.63} C_VEL
LIN {X 0,Y 296.342,Z 669.115,A -85,B 0,C 180,E1 -16453.465,E2 -16453.465} C_VEL
LIN {X 0,Y 296.363,Z 669.318,A -85,B 0,C 180,E1 -16456.482,E2 -16456.482} C_VEL
LIN {X 0,Y 296.313,Z 668.627,A -85,B 0,C 180,E1 -16459.062,E2 -16459.062} C_VEL
LIN {X 0,Y 296.461,Z 666.878,A -85,B 0,C 180,E1 -16461.822,E2 -16461.822} C_VEL
LIN {X 0,Y 296.827,Z 664.204,A -85,B 0,C 180,E1 -16464.565,E2 -16464.565} C_VEL
LIN {X 0,Y 297.446,Z 659.374,A -85,B 0,C 180,E1 -16467.969,E2 -16467.969} C_VEL
LIN {X 0,Y 298.231,Z 654.277,A -85,B 0,C 180,E1 -16470.675,E2 -16470.675} C_VEL
LIN {X 0,Y 299.468,Z 648.077,A -85,B 0,C 180,E1 -16473.363,E2 -16473.363} C_VEL
LIN {X 0,Y 301.318,Z 639.538,A -85,B 0,C 180,E1 -16476.361,E2 -16476.361} C_VEL
LIN {X 0,Y 303.634,Z 630.305,A -85,B 0,C 180,E1 -16478.988,E2 -16478.988} C_VEL
LIN {X 0,Y 305.974,Z 620.821,A -85,B 0,C 180,E1 -16481.259,E2 -16481.259} C_VEL
LIN {X 0,Y 308.582,Z 609.817,A -85,B 0,C 180,E1 -16483.5,E2 -16483.5} C_VEL
LIN {X 0,Y 311.074,Z 598.824,A -85,B 0,C 180,E1 -16485.394,E2 -16485.394} C_VEL
LIN {X 0,Y 313.881,Z 585.952,A -85,B 0,C 180,E1 -16487.258,E2 -16487.258} C_VEL
LIN {X 0,Y 316.749,Z 572.011,A -85,B 0,C 180,E1 -16488.935,E2 -16488.935} C_VEL
LIN {X 0,Y 319.244,Z 558.528,A -85,B 0,C 180,E1 -16490.287,E2 -16490.287} C_VEL
LIN {X 0,Y 321.545,Z 543.953,A -85,B 0,C 180,E1 -16491.475,E2 -16491.475} C_VEL
LIN {X 0,Y 323.264,Z 530.68,A -85,B 0,C 180,E1 -16492.362,E2 -16492.362} C_VEL
LIN {X 0,Y 325.093,Z 514.489,A -85,B 0,C 180,E1 -16493.195,E2 -16493.195} C_VEL
LIN {X 0,Y 326.525,Z 497.548,A -85,B 0,C 180,E1 -16493.801,E2 -16493.801} C_VEL
LIN {X 0,Y 328.229,Z 456.683,A -85,B 0,C 180,E1 -16494.721,E2 -16494.721} C_VEL
LIN {X 0,Y 331.992,Z 361.383,A -85,B 0,C 180,E1 -16496.764,E2 -16496.764} C_VEL
LIN {X 0,Y 331.418,Z 358.442,A -85,B 0,C 180,E1 -16496.913,E2 -16496.913} C_VEL
LIN {X 0,Y 329.881,Z 356.011,A -85,B 0,C 180,E1 -16497.171,E2 -16497.171} C_VEL
LIN {X 0,Y 327.423,Z 353.688,A -85,B 0,C 180,E1 -16497.545,E2 -16497.545} C_VEL
LIN {X 0,Y 322.741,Z 349.912,A -85,B 0,C 180,E1 -16498.261,E2 -16498.261} C_VEL
LIN {X 0,Y 320.588,Z 346.888,A -85,B 0,C 180,E1 -16498.635,E2 -16498.635} C_VEL
LIN {X 0,Y 310.715,Z 329.311,A -85,B 0,C 180,E1 -16500.552,E2 -16500.552} C_VEL
LIN {X 0,Y 301.219,Z 314.236,A -85,B 0,C 180,E1 -16502.501,E2 -16502.501} C_VEL
LIN {X 0,Y 296.171,Z 306.681,A -85,B 0,C 180,E1 -16503.598,E2 -16503.598} C_VEL
LIN {X 0,Y 293.886,Z 303.093,A -85,B 0,C 180,E1 -16504.117,E2 -16504.117} C_VEL
LIN {X 0,Y 292.12,Z 300.826,A -85,B 0,C 180,E1 -16504.509,E2 -16504.509} C_VEL
LIN {X 0,Y 291.394,Z 298.492,A -85,B 0,C 180,E1 -16504.732,E2 -16504.732} C_VEL
LIN {X 0,Y 291.355,Z 298.501,A -85,B 0,C 180,E1 -16507.247,E2 -16507.247} C_VEL
LIN {X 0,Y 291.302,Z 298.51,A -85,B 0,C 180,E1 -16510.648,E2 -16510.648} C_VEL
LIN {X 0,Y 291.284,Z 298.514,A -85,B 0,C 180,E1 -16514.403,E2 -16514.403} C_VEL
LIN {X 0,Y 291.296,Z 298.512,A -85,B 0,C 180,E1 -16518.411,E2 -16518.411} C_VEL
LIN {X 0,Y 291.355,Z 298.446,A -85,B 0,C 180,E1 -16522.751,E2 -16522.751} C_VEL
LIN {X 0,Y 291.345,Z 298.486,A -85,B 0,C 180,E1 -16526.301,E2 -16526.301} C_VEL
LIN {X 0,Y 291.336,Z 298.49,A -85,B 0,C 180,E1 -16530.278,E2 -16530.278} C_VEL
LIN {X 0,Y 291.359,Z 298.501,A -85,B 0,C 180,E1 -16534.266,E2 -16534.266} C_VEL
LIN {X 0,Y 291.366,Z 298.49,A -85,B 0,C 180,E1 -16537.297,E2 -16537.297} C_VEL
LIN {X 0,Y 291.441,Z 298.489,A -85,B 0,C 180,E1 -16540.268,E2 -16540.268} C_VEL
LIN {X 0,Y 291.516,Z 298.484,A -85,B 0,C 180,E1 -16544.652,E2 -16544.652} C_VEL
LIN {X 0,Y 291.536,Z 298.464,A -85,B 0,C 180,E1 -16548.88,E2 -16548.88} C_VEL
LIN {X 0,Y 291.668,Z 298.465,A -85,B 0,C 180,E1 -16551.687,E2 -16551.687} C_VEL
LIN {X 0,Y 291.616,Z 298.451,A -85,B 0,C 180,E1 -16554.467,E2 -16554.467} C_VEL
LIN {X 0,Y 291.886,Z 298.433,A -85,B 0,C 180,E1 -16558.62,E2 -16558.62} C_VEL
LIN {X 0,Y 291.888,Z 298.421,A -85,B 0,C 180,E1 -16561.379,E2 -16561.379} C_VEL
LIN {X 0,Y 291.727,Z 298.428,A -85,B 0,C 180,E1 -16566.918,E2 -16566.918} C_VEL
LIN {X 0,Y 291.575,Z 298.473,A -85,B 0,C 180,E1 -16569.713,E2 -16569.713} C_VEL
LIN {X 0,Y 291.515,Z 298.486,A -85,B 0,C 180,E1 -16573.95,E2 -16573.95} C_VEL
LIN {X 0,Y 291.448,Z 298.494,A -85,B 0,C 180,E1 -16578.269,E2 -16578.269} C_VEL
LIN {X 0,Y 291.373,Z 298.504,A -85,B 0,C 180,E1 -16581.21,E2 -16581.21} C_VEL
LIN {X 0,Y 291.399,Z 298.502,A -85,B 0,C 180,E1 -16584.205,E2 -16584.205} C_VEL
LIN {X 0,Y 291.419,Z 298.497,A -85,B 0,C 180,E1 -16587.271,E2 -16587.271} C_VEL
LIN {X 0,Y 291.332,Z 298.507,A -85,B 0,C 180,E1 -16590.437,E2 -16590.437} C_VEL
LIN {X 0,Y 291.343,Z 298.505,A -85,B 0,C 180,E1 -16593.698,E2 -16593.698} C_VEL
LIN {X 0,Y 291.379,Z 298.486,A -85,B 0,C 180,E1 -16597.255,E2 -16597.255} C_VEL
LIN {X 0,Y 291.369,Z 298.547,A -85,B 0,C 180,E1 -16601.006,E2 -16601.006} C_VEL
LIN {X 0,Y 291.747,Z 300.133,A -85,B 0,C 180,E1 -16601.419,E2 -16601.419} C_VEL
LIN {X 0,Y 293.327,Z 303.862,A -85,B 0,C 180,E1 -16602.423,E2 -16602.423} C_VEL
LIN {X 0,Y 302.617,Z 319.24,A -85,B 0,C 180,E1 -16604.499,E2 -16604.499} C_VEL
LIN {X 0,Y 311.723,Z 335.922,A -85,B 0,C 180,E1 -16606.408,E2 -16606.408} C_VEL
LIN {X 0,Y 320.908,Z 354.827,A -85,B 0,C 180,E1 -16608.242,E2 -16608.242} C_VEL
LIN {X 0,Y 326.147,Z 366.586,A -85,B 0,C 180,E1 -16609.253,E2 -16609.253} C_VEL
LIN {X 0,Y 320.851,Z 499.999,A -85,B 0,C 180,E1 -16612.17,E2 -16612.17} C_VEL
LIN {X 0,Y 319.893,Z 517.31,A -85,B 0,C 180,E1 -16612.633,E2 -16612.633} C_VEL
LIN {X 0,Y 318.225,Z 534.19,A -85,B 0,C 180,E1 -16613.297,E2 -16613.297} C_VEL
LIN {X 0,Y 316.266,Z 549.457,A -85,B 0,C 180,E1 -16614.119,E2 -16614.119} C_VEL
LIN {X 0,Y 313.946,Z 564.59,A -85,B 0,C 180,E1 -16615.191,E2 -16615.191} C_VEL
LIN {X 0,Y 311.296,Z 578.687,A -85,B 0,C 180,E1 -16616.419,E2 -16616.419} C_VEL
LIN {X 0,Y 308.375,Z 593.405,A -85,B 0,C 180,E1 -16618.003,E2 -16618.003} C_VEL
LIN {X 0,Y 305.556,Z 605.863,A -85,B 0,C 180,E1 -16619.601,E2 -16619.601} C_VEL
LIN {X 0,Y 302.568,Z 618.544,A -85,B 0,C 180,E1 -16621.564,E2 -16621.564} C_VEL
LIN {X 0,Y 299.946,Z 629.469,A -85,B 0,C 180,E1 -16623.565,E2 -16623.565} C_VEL
LIN {X 0,Y 297.232,Z 640.437,A -85,B 0,C 180,E1 -16625.929,E2 -16625.929} C_VEL
LIN {X 0,Y 294.868,Z 650.355,A -85,B 0,C 180,E1 -16628.5,E2 -16628.5} C_VEL
LIN {X 0,Y 293.007,Z 658.747,A -85,B 0,C 180,E1 -16631.107,E2 -16631.107} C_VEL
LIN {X 0,Y 291.463,Z 666.266,A -85,B 0,C 180,E1 -16633.901,E2 -16633.901} C_VEL
LIN {X 0,Y 290.434,Z 672.443,A -85,B 0,C 180,E1 -16636.71,E2 -16636.71} C_VEL
LIN {X 0,Y 289.754,Z 677.357,A -85,B 0,C 180,E1 -16639.519,E2 -16639.519} C_VEL
LIN {X 0,Y 289.535,Z 680.33,A -85,B 0,C 180,E1 -16641.626,E2 -16641.626} C_VEL
LIN {X 0,Y 289.474,Z 683.428,A -85,B 0,C 180,E1 -16644.508,E2 -16644.508} C_VEL
LIN {X 0,Y 289.452,Z 685.327,A -85,B 0,C 180,E1 -16647.217,E2 -16647.217} C_VEL
LIN {X 0,Y 289.434,Z 686.317,A -85,B 0,C 180,E1 -16650,E2 -16650} C_VEL
LIN {X 0,Y 289.419,Z 686.307,A -85,B 0,C 180,E1 -16652.784,E2 -16652.784} C_VEL
LIN {X 0,Y 289.429,Z 685.359,A -85,B 0,C 180,E1 -16655.574,E2 -16655.574} C_VEL
LIN {X 0,Y 289.544,Z 683.415,A -85,B 0,C 180,E1 -16658.374,E2 -16658.374} C_VEL
LIN {X 0,Y 289.949,Z 680.523,A -85,B 0,C 180,E1 -16661.181,E2 -16661.181} C_VEL
LIN {X 0,Y 290.884,Z 676.585,A -85,B 0,C 180,E1 -16663.982,E2 -16663.982} C_VEL
LIN {X 0,Y 292.128,Z 671.593,A -85,B 0,C 180,E1 -16666.78,E2 -16666.78} C_VEL
LIN {X 0,Y 294.045,Z 665.474,A -85,B 0,C 180,E1 -16669.549,E2 -16669.549} C_VEL
LIN {X 0,Y 296.651,Z 657.45,A -85,B 0,C 180,E1 -16672.49,E2 -16672.49} C_VEL
LIN {X 0,Y 299.92,Z 648.001,A -85,B 0,C 180,E1 -16675.319,E2 -16675.319} C_VEL
LIN {X 0,Y 303.615,Z 637.487,A -85,B 0,C 180,E1 -16677.907,E2 -16677.907} C_VEL
LIN {X 0,Y 307.381,Z 626.336,A -85,B 0,C 180,E1 -16680.2,E2 -16680.2} C_VEL
LIN {X 0,Y 311.587,Z 613.402,A -85,B 0,C 180,E1 -16682.391,E2 -16682.391} C_VEL
LIN {X 0,Y 315.479,Z 600.989,A -85,B 0,C 180,E1 -16684.106,E2 -16684.106} C_VEL
LIN {X 0,Y 318.869,Z 588.828,A -85,B 0,C 180,E1 -16685.543,E2 -16685.543} C_VEL
LIN {X 0,Y 322.734,Z 573.888,A -85,B 0,C 180,E1 -16686.983,E2 -16686.983} C_VEL
LIN {X 0,Y 325.963,Z 559.266,A -85,B 0,C 180,E1 -16688.11,E2 -16688.11} C_VEL
LIN {X 0,Y 328.608,Z 544.703,A -85,B 0,C 180,E1 -16689.02,E2 -16689.02} C_VEL
LIN {X 0,Y 331.087,Z 528.744,A -85,B 0,C 180,E1 -16689.763,E2 -16689.763} C_VEL
LIN {X 0,Y 332.948,Z 512.008,A -85,B 0,C 180,E1 -16690.318,E2 -16690.318} C_VEL
LIN {X 0,Y 337.101,Z 432.057,A -85,B 0,C 180,E1 -16692.073,E2 -16692.073} C_VEL
LIN {X 0,Y 339.961,Z 375.076,A -85,B 0,C 180,E1 -16693.311,E2 -16693.311} C_VEL
LIN {X 0,Y 331.876,Z 359.237,A -85,B 0,C 180,E1 -16695.402,E2 -16695.402} C_VEL
LIN {X 0,Y 324.138,Z 345.851,A -85,B 0,C 180,E1 -16697.54,E2 -16697.54} C_VEL
LIN {X 0,Y 316.66,Z 334.161,A -85,B 0,C 180,E1 -16699.782,E2 -16699.782} C_VEL
LIN {X 0,Y 310.459,Z 325.073,A -85,B 0,C 180,E1 -16701.81,E2 -16701.81} C_VEL
LIN {X 0,Y 304.51,Z 316.835,A -85,B 0,C 180,E1 -16703.936,E2 -16703.936} C_VEL
LIN {X 0,Y 301.164,Z 312.341,A -85,B 0,C 180,E1 -16705.231,E2 -16705.231} C_VEL
LIN {X 0,Y 298.518,Z 308.911,A -85,B 0,C 180,E1 -16706.31,E2 -16706.31} C_VEL
LIN {X 0,Y 297.422,Z 307.404,A -85,B 0,C 180,E1 -16706.777,E2 -16706.777} C_VEL
LIN {X 0,Y 294.756,Z 304.261,A -85,B 0,C 180,E1 -16707.934,E2 -16707.934} C_VEL
LIN {X 0,Y 293.49,Z 302.715,A -85,B 0,C 180,E1 -16708.512,E2 -16708.512} C_VEL
LIN {X 0,Y 292.083,Z 300.845,A -85,B 0,C 180,E1 -16709.25,E2 -16709.25} C_VEL
LIN {X 0,Y 291.395,Z 298.48,A -85,B 0,C 180,E1 -16710.473,E2 -16710.473} C_VEL
LIN {X 0,Y 291.415,Z 298.496,A -85,B 0,C 180,E1 -16714.273,E2 -16714.273} C_VEL
LIN {X 0,Y 291.374,Z 298.468,A -85,B 0,C 180,E1 -16717.3,E2 -16717.3} C_VEL
LIN {X 0,Y 291.459,Z 298.494,A -85,B 0,C 180,E1 -16720.271,E2 -16720.271} C_VEL
LIN {X 0,Y 291.556,Z 298.454,A -85,B 0,C 180,E1 -16724.625,E2 -16724.625} C_VEL
LIN {X 0,Y 291.53,Z 298.445,A -85,B 0,C 180,E1 -16728.881,E2 -16728.881} C_VEL
LIN {X 0,Y 291.653,Z 298.458,A -85,B 0,C 180,E1 -16731.688,E2 -16731.688} C_VEL
LIN {X 0,Y 291.606,Z 298.441,A -85,B 0,C 180,E1 -16734.469,E2 -16734.469} C_VEL
LIN {X 0,Y 291.884,Z 298.44,A -85,B 0,C 180,E1 -16738.621,E2 -16738.621} C_VEL
LIN {X 0,Y 291.881,Z 298.402,A -85,B 0,C 180,E1 -16741.38,E2 -16741.38} C_VEL
LIN {X 0,Y 291.689,Z 298.434,A -85,B 0,C 180,E1 -16746.92,E2 -16746.92} C_VEL
LIN {X 0,Y 291.57,Z 298.456,A -85,B 0,C 180,E1 -16749.715,E2 -16749.715} C_VEL
LIN {X 0,Y 291.516,Z 298.451,A -85,B 0,C 180,E1 -16753.951,E2 -16753.951} C_VEL
LIN {X 0,Y 291.443,Z 298.614,A -85,B 0,C 180,E1 -16757.862,E2 -16757.862} C_VEL
LIN {X 0,Y 292.126,Z 300.792,A -85,B 0,C 180,E1 -16758.272,E2 -16758.272} C_VEL
LIN {X 0,Y 293.885,Z 303.026,A -85,B 0,C 180,E1 -16759.107,E2 -16759.107} C_VEL
LIN {X 0,Y 296.024,Z 304.486,A -85,B 0,C 180,E1 -16760.005,E2 -16760.005} C_VEL
LIN {X 0,Y 297.728,Z 307.474,A -85,B 0,C 180,E1 -16760.783,E2 -16760.783} C_VEL
LIN {X 0,Y 300.52,Z 309.988,A -85,B 0,C 180,E1 -16761.884,E2 -16761.884} C_VEL
LIN {X 0,Y 302.742,Z 313.334,A -85,B 0,C 180,E1 -16762.783,E2 -16762.783} C_VEL
LIN {X 0,Y 304.939,Z 315.587,A -85,B 0,C 180,E1 -16763.588,E2 -16763.588} C_VEL
LIN {X 0,Y 307.807,Z 319.293,A -85,B 0,C 180,E1 -16764.627,E2 -16764.627} C_VEL
LIN {X 0,Y 309.58,Z 321.626,A -85,B 0,C 180,E1 -16765.243,E2 -16765.243} C_VEL
LIN {X 0,Y 312.99,Z 325.966,A -85,B 0,C 180,E1 -16766.373,E2 -16766.373} C_VEL
LIN {X 0,Y 316.886,Z 331.224,A -85,B 0,C 180,E1 -16767.608,E2 -16767.608} C_VEL
LIN {X 0,Y 321.852,Z 337.963,A -85,B 0,C 180,E1 -16769.089,E2 -16769.089} C_VEL
LIN {X 0,Y 330.104,Z 350.229,A -85,B 0,C 180,E1 -16771.37,E2 -16771.37} C_VEL
LIN {X 0,Y 335.341,Z 358.876,A -85,B 0,C 180,E1 -16772.734,E2 -16772.734} C_VEL
LIN {X 0,Y 340.277,Z 368.267,A -85,B 0,C 180,E1 -16773.982,E2 -16773.982} C_VEL
LIN {X 0,Y 333.572,Z 496.946,A -85,B 0,C 180,E1 -16776.772,E2 -16776.772} C_VEL
LIN {X 0,Y 331.978,Z 512.648,A -85,B 0,C 180,E1 -16777.294,E2 -16777.294} C_VEL
LIN {X 0,Y 329.809,Z 528.776,A -85,B 0,C 180,E1 -16778.059,E2 -16778.059} C_VEL
LIN {X 0,Y 327.242,Z 543.765,A -85,B 0,C 180,E1 -16778.988,E2 -16778.988} C_VEL
LIN {X 0,Y 324.145,Z 558.643,A -85,B 0,C 180,E1 -16780.157,E2 -16780.157} C_VEL
LIN {X 0,Y 320.47,Z 573.64,A -85,B 0,C 180,E1 -16781.622,E2 -16781.622} C_VEL
LIN {X 0,Y 316.753,Z 586.992,A -85,B 0,C 180,E1 -16783.213,E2 -16783.213} C_VEL
LIN {X 0,Y 313.048,Z 599.383,A -85,B 0,C 180,E1 -16784.994,E2 -16784.994} C_VEL
LIN {X 0,Y 309.195,Z 611.123,A -85,B 0,C 180,E1 -16787.007,E2 -16787.007} C_VEL
LIN {X 0,Y 305.2,Z 622.511,A -85,B 0,C 180,E1 -16789.364,E2 -16789.364} C_VEL
LIN {X 0,Y 301.572,Z 632.516,A -85,B 0,C 180,E1 -16791.861,E2 -16791.861} C_VEL
LIN {X 0,Y 298.589,Z 640.883,A -85,B 0,C 180,E1 -16794.37,E2 -16794.37} C_VEL
LIN {X 0,Y 296.047,Z 647.896,A -85,B 0,C 180,E1 -16796.906,E2 -16796.906} C_VEL
LIN {X 0,Y 293.716,Z 654.528,A -85,B 0,C 180,E1 -16799.835,E2 -16799.835} C_VEL
LIN {X 0,Y 291.872,Z 660.173,A -85,B 0,C 180,E1 -16802.991,E2 -16802.991} C_VEL
LIN {X 0,Y 290.728,Z 663.922,A -85,B 0,C 180,E1 -16805.735,E2 -16805.735} C_VEL
LIN {X 0,Y 289.892,Z 666.851,A -85,B 0,C 180,E1 -16808.675,E2 -16808.675} C_VEL
LIN {X 0,Y 289.477,Z 668.738,A -85,B 0,C 180,E1 -16811.602,E2 -16811.602} C_VEL
LIN {X 0,Y 289.234,Z 669.53,A -85,B 0,C 180,E1 -16814.497,E2 -16814.497} C_VEL
LIN {X 0,Y 289.25,Z 669.399,A -85,B 0,C 180,E1 -16817.369,E2 -16817.369} C_VEL
LIN {X 0,Y 289.256,Z 668.199,A -85,B 0,C 180,E1 -16820.207,E2 -16820.207} C_VEL
LIN {X 0,Y 289.513,Z 666.103,A -85,B 0,C 180,E1 -16823.028,E2 -16823.028} C_VEL
LIN {X 0,Y 289.896,Z 662.926,A -85,B 0,C 180,E1 -16825.829,E2 -16825.829} C_VEL
LIN {X 0,Y 290.503,Z 658.781,A -85,B 0,C 180,E1 -16828.614,E2 -16828.614} C_VEL
LIN {X 0,Y 291.379,Z 653.517,A -85,B 0,C 180,E1 -16831.382,E2 -16831.382} C_VEL
LIN {X 0,Y 292.761,Z 647.057,A -85,B 0,C 180,E1 -16834.13,E2 -16834.13} C_VEL
LIN {X 0,Y 294.572,Z 639.333,A -85,B 0,C 180,E1 -16836.851,E2 -16836.851} C_VEL
LIN {X 0,Y 296.972,Z 630.055,A -85,B 0,C 180,E1 -16839.535,E2 -16839.535} C_VEL
LIN {X 0,Y 299.442,Z 620.468,A -85,B 0,C 180,E1 -16841.851,E2 -16841.851} C_VEL
LIN {X 0,Y 302.173,Z 609.344,A -85,B 0,C 180,E1 -16844.135,E2 -16844.135} C_VEL
LIN {X 0,Y 304.992,Z 597.286,A -85,B 0,C 180,E1 -16846.224,E2 -16846.224} C_VEL
LIN {X 0,Y 307.918,Z 584.112,A -85,B 0,C 180,E1 -16848.118,E2 -16848.118} C_VEL
LIN {X 0,Y 310.694,Z 571.117,A -85,B 0,C 180,E1 -16849.662,E2 -16849.662} C_VEL
LIN {X 0,Y 313.57,Z 555.645,A -85,B 0,C 180,E1 -16851.187,E2 -16851.187} C_VEL
LIN {X 0,Y 315.851,Z 540.554,A -85,B 0,C 180,E1 -16852.398,E2 -16852.398} C_VEL
LIN {X 0,Y 318.018,Z 525.019,A -85,B 0,C 180,E1 -16853.354,E2 -16853.354} C_VEL
LIN {X 0,Y 319.522,Z 510.087,A -85,B 0,C 180,E1 -16854.054,E2 -16854.054} C_VEL
LIN {X 0,Y 320.791,Z 493.447,A -85,B 0,C 180,E1 -16854.598,E2 -16854.598} C_VEL
LIN {X 0,Y 326.355,Z 359.509,A -85,B 0,C 180,E1 -16857.526,E2 -16857.526} C_VEL
LIN {X 0,Y 320.588,Z 346.888,A -85,B 0,C 180,E1 -16858.635,E2 -16858.635} C_VEL
LIN {X 0,Y 318.786,Z 343.908,A -85,B 0,C 180,E1 -16858.967,E2 -16858.967} C_VEL
LIN {X 0,Y 316.557,Z 341.418,A -85,B 0,C 180,E1 -16859.35,E2 -16859.35} C_VEL
LIN {X 0,Y 305.295,Z 332.071,A -85,B 0,C 180,E1 -16861.298,E2 -16861.298} C_VEL
LIN {X 0,Y 302.469,Z 327.846,A -85,B 0,C 180,E1 -16861.874,E2 -16861.874} C_VEL
LIN {X 0,Y 294.361,Z 315.202,A -85,B 0,C 180,E1 -16863.638,E2 -16863.638} C_VEL
LIN {X 0,Y 289.533,Z 307.996,A -85,B 0,C 180,E1 -16864.742,E2 -16864.742} C_VEL
LIN {X 0,Y 287.45,Z 304.743,A -85,B 0,C 180,E1 -16865.241,E2 -16865.241} C_VEL
LIN {X 0,Y 284.982,Z 301.602,A -85,B 0,C 180,E1 -16865.822,E2 -16865.822} C_VEL
LIN {X 0,Y 284.316,Z 299.379,A -85,B 0,C 180,E1 -16866.043,E2 -16866.043} C_VEL
LIN {X 0,Y 284.284,Z 299.387,A -85,B 0,C 180,E1 -16869.998,E2 -16869.998} C_VEL
LIN {X 0,Y 284.236,Z 299.393,A -85,B 0,C 180,E1 -16874.187,E2 -16874.187} C_VEL
LIN {X 0,Y 284.241,Z 299.387,A -85,B 0,C 180,E1 -16878.118,E2 -16878.118} C_VEL
LIN {X 0,Y 284.284,Z 299.329,A -85,B 0,C 180,E1 -16882.288,E2 -16882.288} C_VEL
LIN {X 0,Y 284.308,Z 299.34,A -85,B 0,C 180,E1 -16885.35,E2 -16885.35} C_VEL
LIN {X 0,Y 284.28,Z 299.385,A -85,B 0,C 180,E1 -16888.723,E2 -16888.723} C_VEL
LIN {X 0,Y 284.327,Z 299.379,A -85,B 0,C 180,E1 -16892.854,E2 -16892.854} C_VEL
LIN {X 0,Y 284.328,Z 299.361,A -85,B 0,C 180,E1 -16896.703,E2 -16896.703} C_VEL
LIN {X 0,Y 284.377,Z 299.372,A -85,B 0,C 180,E1 -16899.904,E2 -16899.904} C_VEL
LIN {X 0,Y 284.456,Z 299.363,A -85,B 0,C 180,E1 -16904.486,E2 -16904.486} C_VEL
LIN {X 0,Y 284.488,Z 299.34,A -85,B 0,C 180,E1 -16908.601,E2 -16908.601} C_VEL
LIN {X 0,Y 284.623,Z 299.345,A -85,B 0,C 180,E1 -16911.479,E2 -16911.479} C_VEL
LIN {X 0,Y 284.586,Z 299.326,A -85,B 0,C 180,E1 -16914.33,E2 -16914.33} C_VEL
LIN {X 0,Y 284.852,Z 299.31,A -85,B 0,C 180,E1 -16918.585,E2 -16918.585} C_VEL
LIN {X 0,Y 284.854,Z 299.297,A -85,B 0,C 180,E1 -16921.413,E2 -16921.413} C_VEL
LIN {X 0,Y 284.68,Z 299.305,A -85,B 0,C 180,E1 -16927.09,E2 -16927.09} C_VEL
LIN {X 0,Y 284.519,Z 299.356,A -85,B 0,C 180,E1 -16929.956,E2 -16929.956} C_VEL
LIN {X 0,Y 284.463,Z 299.364,A -85,B 0,C 180,E1 -16934.303,E2 -16934.303} C_VEL
LIN {X 0,Y 284.385,Z 299.371,A -85,B 0,C 180,E1 -16938.739,E2 -16938.739} C_VEL
LIN {X 0,Y 284.366,Z 299.378,A -85,B 0,C 180,E1 -16943.292,E2 -16943.292} C_VEL
LIN {X 0,Y 284.394,Z 299.373,A -85,B 0,C 180,E1 -16947.172,E2 -16947.172} C_VEL
LIN {X 0,Y 284.292,Z 299.384,A -85,B 0,C 180,E1 -16951.274,E2 -16951.274} C_VEL
LIN {X 0,Y 284.339,Z 299.371,A -85,B 0,C 180,E1 -16955.348,E2 -16955.348} C_VEL
LIN {X 0,Y 284.336,Z 299.375,A -85,B 0,C 180,E1 -16959.528,E2 -16959.528} C_VEL
LIN {X 0,Y 284.355,Z 299.564,A -85,B 0,C 180,E1 -16959.919,E2 -16959.919} C_VEL
LIN {X 0,Y 285.794,Z 303.477,A -85,B 0,C 180,E1 -16961.015,E2 -16961.015} C_VEL
LIN {X 0,Y 295.379,Z 319.015,A -85,B 0,C 180,E1 -16963.277,E2 -16963.277} C_VEL
LIN {X 0,Y 302.992,Z 332.53,A -85,B 0,C 180,E1 -16964.969,E2 -16964.969} C_VEL
LIN {X 0,Y 311.157,Z 348.57,A -85,B 0,C 180,E1 -16966.694,E2 -16966.694} C_VEL
LIN {X 0,Y 319.71,Z 367.271,A -85,B 0,C 180,E1 -16968.427,E2 -16968.427} C_VEL
LIN {X 0,Y 320.429,Z 368.941,A -85,B 0,C 180,E1 -16968.569,E2 -16968.569} C_VEL
LIN {X 0,Y 314.432,Z 511.017,A -85,B 0,C 180,E1 -16971.738,E2 -16971.738} C_VEL
LIN {X 0,Y 313.024,Z 527.282,A -85,B 0,C 180,E1 -16972.303,E2 -16972.303} C_VEL
LIN {X 0,Y 310.949,Z 543.766,A -85,B 0,C 180,E1 -16973.105,E2 -16973.105} C_VEL
LIN {X 0,Y 308.709,Z 559.112,A -85,B 0,C 180,E1 -16974.111,E2 -16974.111} C_VEL
LIN {X 0,Y 305.931,Z 574.238,A -85,B 0,C 180,E1 -16975.35,E2 -16975.35} C_VEL
LIN {X 0,Y 303.099,Z 588.351,A -85,B 0,C 180,E1 -16976.805,E2 -16976.805} C_VEL
LIN {X 0,Y 299.843,Z 602.528,A -85,B 0,C 180,E1 -16978.566,E2 -16978.566} C_VEL
LIN {X 0,Y 296.762,Z 615.745,A -85,B 0,C 180,E1 -16980.567,E2 -16980.567} C_VEL
LIN {X 0,Y 293.756,Z 627.544,A -85,B 0,C 180,E1 -16982.683,E2 -16982.683} C_VEL
LIN {X 0,Y 290.992,Z 638.292,A -85,B 0,C 180,E1 -16984.998,E2 -16984.998} C_VEL
LIN {X 0,Y 288.427,Z 648.54,A -85,B 0,C 180,E1 -16987.628,E2 -16987.628} C_VEL
LIN {X 0,Y 286.175,Z 658.235,A -85,B 0,C 180,E1 -16990.638,E2 -16990.638} C_VEL
LIN {X 0,Y 284.518,Z 665.819,A -85,B 0,C 180,E1 -16993.497,E2 -16993.497} C_VEL
LIN {X 0,Y 283.445,Z 672.028,A -85,B 0,C 180,E1 -16996.376,E2 -16996.376} C_VEL
LIN {X 0,Y 282.707,Z 676.994,A -85,B 0,C 180,E1 -16999.255,E2 -16999.255} C_VEL
LIN {X 0,Y 282.444,Z 679.992,A -85,B 0,C 180,E1 -17001.414,E2 -17001.414} C_VEL
LIN {X 0,Y 282.395,Z 683.282,A -85,B 0,C 180,E1 -17004.547,E2 -17004.547} C_VEL
LIN {X 0,Y 282.357,Z 685.062,A -85,B 0,C 180,E1 -17007.147,E2 -17007.147} C_VEL
LIN {X 0,Y 282.354,Z 686.098,A -85,B 0,C 180,E1 -17010,E2 -17010} C_VEL
LIN {X 0,Y 282.324,Z 686.11,A -85,B 0,C 180,E1 -17012.854,E2 -17012.854} C_VEL
LIN {X 0,Y 282.332,Z 685.206,A -85,B 0,C 180,E1 -17015.715,E2 -17015.715} C_VEL
LIN {X 0,Y 282.483,Z 683.286,A -85,B 0,C 180,E1 -17018.585,E2 -17018.585} C_VEL
LIN {X 0,Y 282.919,Z 680.444,A -85,B 0,C 180,E1 -17021.463,E2 -17021.463} C_VEL
LIN {X 0,Y 283.931,Z 676.535,A -85,B 0,C 180,E1 -17024.331,E2 -17024.331} C_VEL
LIN {X 0,Y 285.252,Z 671.596,A -85,B 0,C 180,E1 -17027.197,E2 -17027.197} C_VEL
LIN {X 0,Y 287.279,Z 665.505,A -85,B 0,C 180,E1 -17030.029,E2 -17030.029} C_VEL
LIN {X 0,Y 289.839,Z 658.028,A -85,B 0,C 180,E1 -17032.867,E2 -17032.867} C_VEL
LIN {X 0,Y 293.025,Z 649.391,A -85,B 0,C 180,E1 -17035.577,E2 -17035.577} C_VEL
LIN {X 0,Y 296.862,Z 639.032,A -85,B 0,C 180,E1 -17038.261,E2 -17038.261} C_VEL
LIN {X 0,Y 300.655,Z 628.298,A -85,B 0,C 180,E1 -17040.559,E2 -17040.559} C_VEL
LIN {X 0,Y 304.919,Z 615.737,A -85,B 0,C 180,E1 -17042.796,E2 -17042.796} C_VEL
LIN {X 0,Y 309.129,Z 603.093,A -85,B 0,C 180,E1 -17044.637,E2 -17044.637} C_VEL
LIN {X 0,Y 313.167,Z 589.505,A -85,B 0,C 180,E1 -17046.292,E2 -17046.292} C_VEL
LIN {X 0,Y 316.743,Z 576.247,A -85,B 0,C 180,E1 -17047.603,E2 -17047.603} C_VEL
LIN {X 0,Y 320.032,Z 562.265,A -85,B 0,C 180,E1 -17048.746,E2 -17048.746} C_VEL
LIN {X 0,Y 322.975,Z 547.421,A -85,B 0,C 180,E1 -17049.733,E2 -17049.733} C_VEL
LIN {X 0,Y 325.795,Z 530.451,A -85,B 0,C 180,E1 -17050.56,E2 -17050.56} C_VEL
LIN {X 0,Y 327.662,Z 514.722,A -85,B 0,C 180,E1 -17051.107,E2 -17051.107} C_VEL
LIN {X 0,Y 328.995,Z 493.477,A -85,B 0,C 180,E1 -17051.635,E2 -17051.635} C_VEL
LIN {X 0,Y 335.081,Z 377.951,A -85,B 0,C 180,E1 -17054.146,E2 -17054.146} C_VEL
LIN {X 0,Y 327.957,Z 363.778,A -85,B 0,C 180,E1 -17056.07,E2 -17056.07} C_VEL
LIN {X 0,Y 320.372,Z 350.531,A -85,B 0,C 180,E1 -17058.245,E2 -17058.245} C_VEL
LIN {X 0,Y 313.276,Z 339.161,A -85,B 0,C 180,E1 -17060.465,E2 -17060.465} C_VEL
LIN {X 0,Y 307.569,Z 330.771,A -85,B 0,C 180,E1 -17062.394,E2 -17062.394} C_VEL
LIN {X 0,Y 302.436,Z 323.452,A -85,B 0,C 180,E1 -17064.291,E2 -17064.291} C_VEL
LIN {X 0,Y 298.85,Z 318.56,A -85,B 0,C 180,E1 -17065.716,E2 -17065.716} C_VEL
LIN {X 0,Y 295.966,Z 314.689,A -85,B 0,C 180,E1 -17066.934,E2 -17066.934} C_VEL
LIN {X 0,Y 292.319,Z 310.076,A -85,B 0,C 180,E1 -17068.574,E2 -17068.574} C_VEL
LIN {X 0,Y 287.889,Z 304.65,A -85,B 0,C 180,E1 -17070.776,E2 -17070.776} C_VEL
LIN {X 0,Y 285.594,Z 302.596,A -85,B 0,C 180,E1 -17071.975,E2 -17071.975} C_VEL
LIN {X 0,Y 284.581,Z 300.394,A -85,B 0,C 180,E1 -17072.643,E2 -17072.643} C_VEL
LIN {X 0,Y 284.397,Z 299.349,A -85,B 0,C 180,E1 -17073.282,E2 -17073.282} C_VEL
LIN {X 0,Y 284.333,Z 299.346,A -85,B 0,C 180,E1 -17076.705,E2 -17076.705} C_VEL
LIN {X 0,Y 284.404,Z 299.353,A -85,B 0,C 180,E1 -17081.262,E2 -17081.262} C_VEL
LIN {X 0,Y 284.493,Z 299.33,A -85,B 0,C 180,E1 -17084.46,E2 -17084.46} C_VEL
LIN {X 0,Y 284.468,Z 299.325,A -85,B 0,C 180,E1 -17088.601,E2 -17088.601} C_VEL
LIN {X 0,Y 284.61,Z 299.329,A -85,B 0,C 180,E1 -17091.48,E2 -17091.48} C_VEL
LIN {X 0,Y 284.575,Z 299.318,A -85,B 0,C 180,E1 -17094.331,E2 -17094.331} C_VEL
LIN {X 0,Y 284.851,Z 299.315,A -85,B 0,C 180,E1 -17098.587,E2 -17098.587} C_VEL
LIN {X 0,Y 284.847,Z 299.277,A -85,B 0,C 180,E1 -17101.415,E2 -17101.415} C_VEL
LIN {X 0,Y 284.645,Z 299.309,A -85,B 0,C 180,E1 -17107.092,E2 -17107.092} C_VEL
LIN {X 0,Y 284.516,Z 299.338,A -85,B 0,C 180,E1 -17109.958,E2 -17109.958} C_VEL
LIN {X 0,Y 284.46,Z 299.331,A -85,B 0,C 180,E1 -17114.305,E2 -17114.305} C_VEL
LIN {X 0,Y 284.461,Z 299.366,A -85,B 0,C 180,E1 -17114.699,E2 -17114.699} C_VEL
LIN {X 0,Y 285.036,Z 301.45,A -85,B 0,C 180,E1 -17115.124,E2 -17115.124} C_VEL
LIN {X 0,Y 286.755,Z 303.793,A -85,B 0,C 180,E1 -17116.097,E2 -17116.097} C_VEL
LIN {X 0,Y 289.251,Z 305.355,A -85,B 0,C 180,E1 -17117.317,E2 -17117.317} C_VEL
LIN {X 0,Y 290.684,Z 308.148,A -85,B 0,C 180,E1 -17118.092,E2 -17118.092} C_VEL
LIN {X 0,Y 293.362,Z 310.558,A -85,B 0,C 180,E1 -17119.313,E2 -17119.313} C_VEL
LIN {X 0,Y 293.983,Z 311.331,A -85,B 0,C 180,E1 -17119.594,E2 -17119.594} C_VEL
LIN {X 0,Y 296.314,Z 314.665,A -85,B 0,C 180,E1 -17120.638,E2 -17120.638} C_VEL
LIN {X 0,Y 298.286,Z 316.488,A -85,B 0,C 180,E1 -17121.432,E2 -17121.432} C_VEL
LIN {X 0,Y 301.018,Z 320.216,A -85,B 0,C 180,E1 -17122.541,E2 -17122.541} C_VEL
LIN {X 0,Y 302.516,Z 321.821,A -85,B 0,C 180,E1 -17123.105,E2 -17123.105} C_VEL
LIN {X 0,Y 305.649,Z 325.773,A -85,B 0,C 180,E1 -17124.265,E2 -17124.265} C_VEL
LIN {X 0,Y 313.137,Z 335.749,A -85,B 0,C 180,E1 -17126.808,E2 -17126.808} C_VEL
LIN {X 0,Y 321.42,Z 347.485,A -85,B 0,C 180,E1 -17129.337,E2 -17129.337} C_VEL
LIN {X 0,Y 329.981,Z 360.872,A -85,B 0,C 180,E1 -17131.705,E2 -17131.705} C_VEL
LIN {X 0,Y 335.297,Z 370.915,A -85,B 0,C 180,E1 -17133.116,E2 -17133.116} C_VEL
LIN {X 0,Y 334.274,Z 391.843,A -85,B 0,C 180,E1 -17133.589,E2 -17133.589} C_VEL
LIN {X 0,Y 328.597,Z 497.064,A -85,B 0,C 180,E1 -17135.897,E2 -17135.897} C_VEL
LIN {X 0,Y 326.955,Z 512.687,A -85,B 0,C 180,E1 -17136.415,E2 -17136.415} C_VEL
LIN {X 0,Y 324.697,Z 529,A -85,B 0,C 180,E1 -17137.195,E2 -17137.195} C_VEL
LIN {X 0,Y 321.89,Z 544.72,A -85,B 0,C 180,E1 -17138.186,E2 -17138.186} C_VEL
LIN {X 0,Y 318.919,Z 558.501,A -85,B 0,C 180,E1 -17139.281,E2 -17139.281} C_VEL
LIN {X 0,Y 315.232,Z 573.095,A -85,B 0,C 180,E1 -17140.71,E2 -17140.71} C_VEL
LIN {X 0,Y 311.515,Z 586.14,A -85,B 0,C 180,E1 -17142.259,E2 -17142.259} C_VEL
LIN {X 0,Y 307.727,Z 598.339,A -85,B 0,C 180,E1 -17143.994,E2 -17143.994} C_VEL
LIN {X 0,Y 303.66,Z 610.201,A -85,B 0,C 180,E1 -17146.026,E2 -17146.026} C_VEL
LIN {X 0,Y 299.384,Z 621.977,A -85,B 0,C 180,E1 -17148.458,E2 -17148.458} C_VEL
LIN {X 0,Y 295.613,Z 631.941,A -85,B 0,C 180,E1 -17150.948,E2 -17150.948} C_VEL
LIN {X 0,Y 292.405,Z 640.435,A -85,B 0,C 180,E1 -17153.496,E2 -17153.496} C_VEL
LIN {X 0,Y 289.699,Z 647.523,A -85,B 0,C 180,E1 -17156.084,E2 -17156.084} C_VEL
LIN {X 0,Y 287.12,Z 654.281,A -85,B 0,C 180,E1 -17159.067,E2 -17159.067} C_VEL
LIN {X 0,Y 285.266,Z 659.727,A -85,B 0,C 180,E1 -17162.089,E2 -17162.089} C_VEL
LIN {X 0,Y 283.85,Z 663.85,A -85,B 0,C 180,E1 -17165.108,E2 -17165.108} C_VEL
LIN {X 0,Y 282.946,Z 666.886,A -85,B 0,C 180,E1 -17168.125,E2 -17168.125} C_VEL
LIN {X 0,Y 282.432,Z 668.823,A -85,B 0,C 180,E1 -17171.126,E2 -17171.126} C_VEL
LIN {X 0,Y 282.142,Z 669.718,A -85,B 0,C 180,E1 -17174.097,E2 -17174.097} C_VEL
LIN {X 0,Y 282.175,Z 669.639,A -85,B 0,C 180,E1 -17177.046,E2 -17177.046} C_VEL
LIN {X 0,Y 282.138,Z 668.535,A -85,B 0,C 180,E1 -17179.958,E2 -17179.958} C_VEL
LIN {X 0,Y 282.408,Z 666.51,A -85,B 0,C 180,E1 -17182.852,E2 -17182.852} C_VEL
LIN {X 0,Y 282.806,Z 663.411,A -85,B 0,C 180,E1 -17185.724,E2 -17185.724} C_VEL
LIN {X 0,Y 283.413,Z 659.371,A -85,B 0,C 180,E1 -17188.579,E2 -17188.579} C_VEL
LIN {X 0,Y 284.636,Z 652.728,A -85,B 0,C 180,E1 -17192.122,E2 -17192.122} C_VEL
LIN {X 0,Y 286.078,Z 646.03,A -85,B 0,C 180,E1 -17194.932,E2 -17194.932} C_VEL
LIN {X 0,Y 288.099,Z 638.007,A -85,B 0,C 180,E1 -17197.71,E2 -17197.71} C_VEL
LIN {X 0,Y 290.706,Z 628.46,A -85,B 0,C 180,E1 -17200.446,E2 -17200.446} C_VEL
LIN {X 0,Y 293.716,Z 617.108,A -85,B 0,C 180,E1 -17203.139,E2 -17203.139} C_VEL
LIN {X 0,Y 296.684,Z 605.359,A -85,B 0,C 180,E1 -17205.456,E2 -17205.456} C_VEL
LIN {X 0,Y 299.515,Z 593.51,A -85,B 0,C 180,E1 -17207.408,E2 -17207.408} C_VEL
LIN {X 0,Y 302.648,Z 579.62,A -85,B 0,C 180,E1 -17209.324,E2 -17209.324} C_VEL
LIN {X 0,Y 305.57,Z 565.863,A -85,B 0,C 180,E1 -17210.885,E2 -17210.885} C_VEL
LIN {X 0,Y 308.211,Z 551.049,A -85,B 0,C 180,E1 -17212.277,E2 -17212.277} C_VEL
LIN {X 0,Y 310.521,Z 535.694,A -85,B 0,C 180,E1 -17213.421,E2 -17213.421} C_VEL
LIN {X 0,Y 312.689,Z 519.243,A -85,B 0,C 180,E1 -17214.349,E2 -17214.349} C_VEL
LIN {X 0,Y 314.266,Z 503.165,A -85,B 0,C 180,E1 -17215.012,E2 -17215.012} C_VEL
LIN {X 0,Y 315.313,Z 485.679,A -85,B 0,C 180,E1 -17215.496,E2 -17215.496} C_VEL
LIN {X 0,Y 320.53,Z 361.607,A -85,B 0,C 180,E1 -17218.234,E2 -17218.234} C_VEL
LIN {X 0,Y 314.098,Z 347.917,A -85,B 0,C 180,E1 -17219.514,E2 -17219.514} C_VEL
LIN {X 0,Y 304.452,Z 331.04,A -85,B 0,C 180,E1 -17221.461,E2 -17221.461} C_VEL
LIN {X 0,Y 302.469,Z 327.846,A -85,B 0,C 180,E1 -17221.874,E2 -17221.874} C_VEL
LIN {X 0,Y 300.716,Z 324.964,A -85,B 0,C 180,E1 -17222.249,E2 -17222.249} C_VEL
LIN {X 0,Y 297.35,Z 321.593,A -85,B 0,C 180,E1 -17222.917,E2 -17222.917} C_VEL
LIN {X 0,Y 287.234,Z 314.589,A -85,B 0,C 180,E1 -17224.947,E2 -17224.947} C_VEL
LIN {X 0,Y 284.044,Z 311.03,A -85,B 0,C 180,E1 -17225.677,E2 -17225.677} C_VEL
LIN {X 0,Y 282.625,Z 308.987,A -85,B 0,C 180,E1 -17226.027,E2 -17226.027} C_VEL
LIN {X 0,Y 280.456,Z 305.628,A -85,B 0,C 180,E1 -17226.58,E2 -17226.58} C_VEL
LIN {X 0,Y 277.965,Z 302.592,A -85,B 0,C 180,E1 -17227.203,E2 -17227.203} C_VEL
LIN {X 0,Y 277.253,Z 300.254,A -85,B 0,C 180,E1 -17227.471,E2 -17227.471} C_VEL
LIN {X 0,Y 277.186,Z 300.26,A -85,B 0,C 180,E1 -17231.241,E2 -17231.241} C_VEL
LIN {X 0,Y 277.176,Z 300.262,A -85,B 0,C 180,E1 -17235.232,E2 -17235.232} C_VEL
LIN {X 0,Y 277.178,Z 300.272,A -85,B 0,C 180,E1 -17238.757,E2 -17238.757} C_VEL
LIN {X 0,Y 277.235,Z 300.203,A -85,B 0,C 180,E1 -17242.524,E2 -17242.524} C_VEL
LIN {X 0,Y 277.247,Z 300.236,A -85,B 0,C 180,E1 -17246.103,E2 -17246.103} C_VEL
LIN {X 0,Y 277.229,Z 300.254,A -85,B 0,C 180,E1 -17249.534,E2 -17249.534} C_VEL
LIN {X 0,Y 277.289,Z 300.255,A -85,B 0,C 180,E1 -17252.856,E2 -17252.856} C_VEL
LIN {X 0,Y 277.283,Z 300.238,A -85,B 0,C 180,E1 -17256.074,E2 -17256.074} C_VEL
LIN {X 0,Y 277.325,Z 300.242,A -85,B 0,C 180,E1 -17260.764,E2 -17260.764} C_VEL
LIN {X 0,Y 277.416,Z 300.243,A -85,B 0,C 180,E1 -17265.324,E2 -17265.324} C_VEL
LIN {X 0,Y 277.461,Z 300.226,A -85,B 0,C 180,E1 -17269.786,E2 -17269.786} C_VEL
LIN {X 0,Y 277.624,Z 300.205,A -85,B 0,C 180,E1 -17272.728,E2 -17272.728} C_VEL
LIN {X 0,Y 277.818,Z 300.186,A -85,B 0,C 180,E1 -17278.55,E2 -17278.55} C_VEL
LIN {X 0,Y 277.82,Z 300.173,A -85,B 0,C 180,E1 -17281.449,E2 -17281.449} C_VEL
LIN {X 0,Y 277.636,Z 300.182,A -85,B 0,C 180,E1 -17287.271,E2 -17287.271} C_VEL
LIN {X 0,Y 277.461,Z 300.235,A -85,B 0,C 180,E1 -17290.212,E2 -17290.212} C_VEL
LIN {X 0,Y 277.409,Z 300.244,A -85,B 0,C 180,E1 -17294.675,E2 -17294.675} C_VEL
LIN {X 0,Y 277.334,Z 300.249,A -85,B 0,C 180,E1 -17299.234,E2 -17299.234} C_VEL
LIN {X 0,Y 277.318,Z 300.257,A -85,B 0,C 180,E1 -17304.17,E2 -17304.17} C_VEL
LIN {X 0,Y 277.322,Z 300.251,A -85,B 0,C 180,E1 -17307.504,E2 -17307.504} C_VEL
LIN {X 0,Y 277.27,Z 300.258,A -85,B 0,C 180,E1 -17310.481,E2 -17310.481} C_VEL
LIN {X 0,Y 277.245,Z 300.261,A -85,B 0,C 180,E1 -17313.895,E2 -17313.895} C_VEL
LIN {X 0,Y 277.27,Z 300.244,A -85,B 0,C 180,E1 -17317.468,E2 -17317.468} C_VEL
LIN {X 0,Y 277.311,Z 300.354,A -85,B 0,C 180,E1 -17318.696,E2 -17318.696} C_VEL
LIN {X 0,Y 278.358,Z 303.205,A -85,B 0,C 180,E1 -17319.518,E2 -17319.518} C_VEL
LIN {X 0,Y 286.939,Z 316.919,A -85,B 0,C 180,E1 -17321.692,E2 -17321.692} C_VEL
LIN {X 0,Y 294.844,Z 330.394,A -85,B 0,C 180,E1 -17323.552,E2 -17323.552} C_VEL
LIN {X 0,Y 303.11,Z 346.048,A -85,B 0,C 180,E1 -17325.401,E2 -17325.401} C_VEL
LIN {X 0,Y 311.707,Z 364.287,A -85,B 0,C 180,E1 -17327.23,E2 -17327.23} C_VEL
LIN {X 0,Y 314.658,Z 371.06,A -85,B 0,C 180,E1 -17327.841,E2 -17327.841} C_VEL
LIN {X 0,Y 308.499,Z 511.722,A -85,B 0,C 180,E1 -17331.029,E2 -17331.029} C_VEL
LIN {X 0,Y 306.95,Z 528.563,A -85,B 0,C 180,E1 -17331.639,E2 -17331.639} C_VEL
LIN {X 0,Y 304.836,Z 544.526,A -85,B 0,C 180,E1 -17332.446,E2 -17332.446} C_VEL
LIN {X 0,Y 302.383,Z 560.673,A -85,B 0,C 180,E1 -17333.55,E2 -17333.55} C_VEL
LIN {X 0,Y 299.343,Z 576.281,A -85,B 0,C 180,E1 -17334.886,E2 -17334.886} C_VEL
LIN {X 0,Y 296.283,Z 590.936,A -85,B 0,C 180,E1 -17336.462,E2 -17336.462} C_VEL
LIN {X 0,Y 292.876,Z 605.19,A -85,B 0,C 180,E1 -17338.337,E2 -17338.337} C_VEL
LIN {X 0,Y 289.93,Z 616.922,A -85,B 0,C 180,E1 -17340.203,E2 -17340.203} C_VEL
LIN {X 0,Y 286.989,Z 628.039,A -85,B 0,C 180,E1 -17342.271,E2 -17342.271} C_VEL
LIN {X 0,Y 284.043,Z 639.142,A -85,B 0,C 180,E1 -17344.735,E2 -17344.735} C_VEL
LIN {X 0,Y 281.287,Z 649.756,A -85,B 0,C 180,E1 -17347.584,E2 -17347.584} C_VEL
LIN {X 0,Y 279.124,Z 658.747,A -85,B 0,C 180,E1 -17350.512,E2 -17350.512} C_VEL
LIN {X 0,Y 277.595,Z 665.361,A -85,B 0,C 180,E1 -17353.073,E2 -17353.073} C_VEL
LIN {X 0,Y 276.459,Z 671.602,A -85,B 0,C 180,E1 -17356.025,E2 -17356.025} C_VEL
LIN {X 0,Y 275.653,Z 676.625,A -85,B 0,C 180,E1 -17358.976,E2 -17358.976} C_VEL
LIN {X 0,Y 275.371,Z 679.65,A -85,B 0,C 180,E1 -17361.192,E2 -17361.192} C_VEL
LIN {X 0,Y 275.312,Z 683.14,A -85,B 0,C 180,E1 -17364.598,E2 -17364.598} C_VEL
LIN {X 0,Y 275.264,Z 684.796,A -85,B 0,C 180,E1 -17367.073,E2 -17367.073} C_VEL
LIN {X 0,Y 275.275,Z 685.879,A -85,B 0,C 180,E1 -17370,E2 -17370} C_VEL
LIN {X 0,Y 275.232,Z 685.914,A -85,B 0,C 180,E1 -17372.928,E2 -17372.928} C_VEL
LIN {X 0,Y 275.227,Z 685.057,A -85,B 0,C 180,E1 -17375.863,E2 -17375.863} C_VEL
LIN {X 0,Y 275.404,Z 683.16,A -85,B 0,C 180,E1 -17378.808,E2 -17378.808} C_VEL
LIN {X 0,Y 275.901,Z 680.368,A -85,B 0,C 180,E1 -17381.758,E2 -17381.758} C_VEL
LIN {X 0,Y 276.973,Z 676.484,A -85,B 0,C 180,E1 -17384.699,E2 -17384.699} C_VEL
LIN {X 0,Y 278.394,Z 671.599,A -85,B 0,C 180,E1 -17387.634,E2 -17387.634} C_VEL
LIN {X 0,Y 280.538,Z 665.54,A -85,B 0,C 180,E1 -17390.532,E2 -17390.532} C_VEL
LIN {X 0,Y 283.192,Z 658.235,A -85,B 0,C 180,E1 -17393.396,E2 -17393.396} C_VEL
LIN {X 0,Y 286.58,Z 649.568,A -85,B 0,C 180,E1 -17396.195,E2 -17396.195} C_VEL
LIN {X 0,Y 290.601,Z 639.267,A -85,B 0,C 180,E1 -17398.927,E2 -17398.927} C_VEL
LIN {X 0,Y 294.525,Z 628.599,A -85,B 0,C 180,E1 -17401.266,E2 -17401.266} C_VEL
LIN {X 0,Y 298.99,Z 616.137,A -85,B 0,C 180,E1 -17403.531,E2 -17403.531} C_VEL
LIN {X 0,Y 303.327,Z 603.629,A -85,B 0,C 180,E1 -17405.398,E2 -17405.398} C_VEL
LIN {X 0,Y 307.499,Z 590.187,A -85,B 0,C 180,E1 -17407.072,E2 -17407.072} C_VEL
LIN {X 0,Y 311.609,Z 575.506,A -85,B 0,C 180,E1 -17408.54,E2 -17408.54} C_VEL
LIN {X 0,Y 315.03,Z 561.386,A -85,B 0,C 180,E1 -17409.687,E2 -17409.687} C_VEL
LIN {X 0,Y 318.093,Z 546.332,A -85,B 0,C 180,E1 -17410.676,E2 -17410.676} C_VEL
LIN {X 0,Y 320.89,Z 529.741,A -85,B 0,C 180,E1 -17411.484,E2 -17411.484} C_VEL
LIN {X 0,Y 322.873,Z 513.338,A -85,B 0,C 180,E1 -17412.045,E2 -17412.045} C_VEL
LIN {X 0,Y 324.418,Z 487.9,A -85,B 0,C 180,E1 -17412.661,E2 -17412.661} C_VEL
LIN {X 0,Y 330.323,Z 380.823,A -85,B 0,C 180,E1 -17415.001,E2 -17415.001} C_VEL
LIN {X 0,Y 323.38,Z 366.997,A -85,B 0,C 180,E1 -17416.958,E2 -17416.958} C_VEL
LIN {X 0,Y 315.788,Z 353.681,A -85,B 0,C 180,E1 -17419.247,E2 -17419.247} C_VEL
LIN {X 0,Y 308.871,Z 342.54,A -85,B 0,C 180,E1 -17421.526,E2 -17421.526} C_VEL
LIN {X 0,Y 301.322,Z 331.394,A -85,B 0,C 180,E1 -17424.281,E2 -17424.281} C_VEL
LIN {X 0,Y 296.666,Z 324.924,A -85,B 0,C 180,E1 -17426.163,E2 -17426.163} C_VEL
LIN {X 0,Y 293.573,Z 320.683,A -85,B 0,C 180,E1 -17427.511,E2 -17427.511} C_VEL
LIN {X 0,Y 290.212,Z 316.355,A -85,B 0,C 180,E1 -17429.08,E2 -17429.08} C_VEL
LIN {X 0,Y 286.104,Z 311.297,A -85,B 0,C 180,E1 -17431.18,E2 -17431.18} C_VEL
LIN {X 0,Y 283.682,Z 308.925,A -85,B 0,C 180,E1 -17432.496,E2 -17432.496} C_VEL
LIN {X 0,Y 282.312,Z 306.239,A -85,B 0,C 180,E1 -17433.379,E2 -17433.379} C_VEL
LIN {X 0,Y 279.234,Z 304.306,A -85,B 0,C 180,E1 -17435.237,E2 -17435.237} C_VEL
LIN {X 0,Y 277.715,Z 301.914,A -85,B 0,C 180,E1 -17436.363,E2 -17436.363} C_VEL
LIN {X 0,Y 277.298,Z 300.221,A -85,B 0,C 180,E1 -17436.82,E2 -17436.82} C_VEL
LIN {X 0,Y 277.345,Z 300.242,A -85,B 0,C 180,E1 -17440.767,E2 -17440.767} C_VEL
LIN {X 0,Y 277.436,Z 300.223,A -85,B 0,C 180,E1 -17445.327,E2 -17445.327} C_VEL
LIN {X 0,Y 277.456,Z 300.196,A -85,B 0,C 180,E1 -17449.788,E2 -17449.788} C_VEL
LIN {X 0,Y 277.603,Z 300.218,A -85,B 0,C 180,E1 -17452.729,E2 -17452.729} C_VEL
LIN {X 0,Y 277.817,Z 300.191,A -85,B 0,C 180,E1 -17458.551,E2 -17458.551} C_VEL
LIN {X 0,Y 277.813,Z 300.152,A -85,B 0,C 180,E1 -17461.45,E2 -17461.45} C_VEL
LIN {X 0,Y 277.603,Z 300.183,A -85,B 0,C 180,E1 -17467.273,E2 -17467.273} C_VEL
LIN {X 0,Y 277.444,Z 300.247,A -85,B 0,C 180,E1 -17470.768,E2 -17470.768} C_VEL
LIN {X 0,Y 278.011,Z 302.271,A -85,B 0,C 180,E1 -17471.299,E2 -17471.299} C_VEL
LIN {X 0,Y 279.586,Z 304.504,A -85,B 0,C 180,E1 -17472.43,E2 -17472.43} C_VEL
LIN {X 0,Y 282.509,Z 306.322,A -85,B 0,C 180,E1 -17474.176,E2 -17474.176} C_VEL
LIN {X 0,Y 284.014,Z 309.255,A -85,B 0,C 180,E1 -17475.137,E2 -17475.137} C_VEL
LIN {X 0,Y 286.568,Z 311.575,A -85,B 0,C 180,E1 -17476.497,E2 -17476.497} C_VEL
LIN {X 0,Y 287.305,Z 312.135,A -85,B 0,C 180,E1 -17476.865,E2 -17476.865} C_VEL
LIN {X 0,Y 289.399,Z 315.384,A -85,B 0,C 180,E1 -17477.969,E2 -17477.969} C_VEL
LIN {X 0,Y 291.776,Z 317.593,A -85,B 0,C 180,E1 -17479.071,E2 -17479.071} C_VEL
LIN {X 0,Y 294.281,Z 321.123,A -85,B 0,C 180,E1 -17480.224,E2 -17480.224} C_VEL
LIN {X 0,Y 296.167,Z 323.055,A -85,B 0,C 180,E1 -17481.012,E2 -17481.012} C_VEL
LIN {X 0,Y 298.975,Z 326.731,A -85,B 0,C 180,E1 -17482.17,E2 -17482.17} C_VEL
LIN {X 0,Y 300.442,Z 328.538,A -85,B 0,C 180,E1 -17482.745,E2 -17482.745} C_VEL
LIN {X 0,Y 304.415,Z 333.745,A -85,B 0,C 180,E1 -17484.243,E2 -17484.243} C_VEL
LIN {X 0,Y 308.436,Z 339.104,A -85,B 0,C 180,E1 -17485.655,E2 -17485.655} C_VEL
LIN {X 0,Y 314.248,Z 347.208,A -85,B 0,C 180,E1 -17487.554,E2 -17487.554} C_VEL
LIN {X 0,Y 321.773,Z 358.528,A -85,B 0,C 180,E1 -17489.821,E2 -17489.821} C_VEL
LIN {X 0,Y 327.68,Z 368.397,A -85,B 0,C 180,E1 -17491.475,E2 -17491.475} C_VEL
LIN {X 0,Y 330.618,Z 374.133,A -85,B 0,C 180,E1 -17492.283,E2 -17492.283} C_VEL
LIN {X 0,Y 323.648,Z 497.787,A -85,B 0,C 180,E1 -17495.009,E2 -17495.009} C_VEL
LIN {X 0,Y 321.905,Z 513.702,A -85,B 0,C 180,E1 -17495.55,E2 -17495.55} C_VEL
LIN {X 0,Y 319.525,Z 530.065,A -85,B 0,C 180,E1 -17496.35,E2 -17496.35} C_VEL
LIN {X 0,Y 316.347,Z 546.646,A -85,B 0,C 180,E1 -17497.418,E2 -17497.418} C_VEL
LIN {X 0,Y 313.09,Z 561.213,A -85,B 0,C 180,E1 -17498.628,E2 -17498.628} C_VEL
LIN {X 0,Y 309.117,Z 576.044,A -85,B 0,C 180,E1 -17500.138,E2 -17500.138} C_VEL
LIN {X 0,Y 304.843,Z 589.958,A -85,B 0,C 180,E1 -17501.888,E2 -17501.888} C_VEL
LIN {X 0,Y 300.69,Z 602.463,A -85,B 0,C 180,E1 -17503.81,E2 -17503.81} C_VEL
LIN {X 0,Y 296.248,Z 614.669,A -85,B 0,C 180,E1 -17506.059,E2 -17506.059} C_VEL
LIN {X 0,Y 292.345,Z 624.816,A -85,B 0,C 180,E1 -17508.296,E2 -17508.296} C_VEL
LIN {X 0,Y 288.084,Z 635.424,A -85,B 0,C 180,E1 -17511.15,E2 -17511.15} C_VEL
LIN {X 0,Y 284.309,Z 644.929,A -85,B 0,C 180,E1 -17514.342,E2 -17514.342} C_VEL
LIN {X 0,Y 281.26,Z 652.448,A -85,B 0,C 180,E1 -17517.504,E2 -17517.504} C_VEL
LIN {X 0,Y 279.028,Z 658.261,A -85,B 0,C 180,E1 -17520.583,E2 -17520.583} C_VEL
LIN {X 0,Y 277.727,Z 661.804,A -85,B 0,C 180,E1 -17522.903,E2 -17522.903} C_VEL
LIN {X 0,Y 276.394,Z 665.732,A -85,B 0,C 180,E1 -17526.263,E2 -17526.263} C_VEL
LIN {X 0,Y 275.648,Z 668.058,A -85,B 0,C 180,E1 -17529.087,E2 -17529.087} C_VEL
LIN {X 0,Y 275.21,Z 669.525,A -85,B 0,C 180,E1 -17532.155,E2 -17532.155} C_VEL
LIN {X 0,Y 275.04,Z 670.046,A -85,B 0,C 180,E1 -17535.195,E2 -17535.195} C_VEL
LIN {X 0,Y 275.038,Z 669.482,A -85,B 0,C 180,E1 -17538.204,E2 -17538.204} C_VEL
LIN {X 0,Y 275.117,Z 668.031,A -85,B 0,C 180,E1 -17541.183,E2 -17541.183} C_VEL
LIN {X 0,Y 275.554,Z 665.5,A -85,B 0,C 180,E1 -17544.144,E2 -17544.144} C_VEL
LIN {X 0,Y 276.129,Z 660.981,A -85,B 0,C 180,E1 -17547.812,E2 -17547.812} C_VEL
LIN {X 0,Y 276.927,Z 656.21,A -85,B 0,C 180,E1 -17550.727,E2 -17550.727} C_VEL
LIN {X 0,Y 278.275,Z 650.228,A -85,B 0,C 180,E1 -17553.62,E2 -17553.62} C_VEL
LIN {X 0,Y 279.997,Z 643.008,A -85,B 0,C 180,E1 -17556.485,E2 -17556.485} C_VEL
LIN {X 0,Y 282.392,Z 634.385,A -85,B 0,C 180,E1 -17559.309,E2 -17559.309} C_VEL
LIN {X 0,Y 285.273,Z 624.126,A -85,B 0,C 180,E1 -17562.087,E2 -17562.087} C_VEL
LIN {X 0,Y 288.143,Z 613.481,A -85,B 0,C 180,E1 -17564.478,E2 -17564.478} C_VEL
LIN {X 0,Y 291.334,Z 601.022,A -85,B 0,C 180,E1 -17566.827,E2 -17566.827} C_VEL
LIN {X 0,Y 294.681,Z 587.306,A -85,B 0,C 180,E1 -17568.962,E2 -17568.962} C_VEL
LIN {X 0,Y 297.827,Z 573.516,A -85,B 0,C 180,E1 -17570.73,E2 -17570.73} C_VEL
LIN {X 0,Y 300.876,Z 558.5,A -85,B 0,C 180,E1 -17572.307,E2 -17572.307} C_VEL
LIN {X 0,Y 303.401,Z 543.836,A -85,B 0,C 180,E1 -17573.552,E2 -17573.552} C_VEL
LIN {X 0,Y 305.541,Z 529.016,A -85,B 0,C 180,E1 -17574.549,E2 -17574.549} C_VEL
LIN {X 0,Y 307.527,Z 511.909,A -85,B 0,C 180,E1 -17575.418,E2 -17575.418} C_VEL
LIN {X 0,Y 308.905,Z 496.119,A -85,B 0,C 180,E1 -17575.974,E2 -17575.974} C_VEL
LIN {X 0,Y 314.747,Z 364.907,A -85,B 0,C 180,E1 -17578.935,E2 -17578.935} C_VEL
LIN {X 0,Y 314.613,Z 363.286,A -85,B 0,C 180,E1 -17579,E2 -17579} C_VEL
LIN {X 0,Y 309.092,Z 351.736,A -85,B 0,C 180,E1 -17580.133,E2 -17580.133} C_VEL
LIN {X 0,Y 299.807,Z 335.372,A -85,B 0,C 180,E1 -17582.072,E2 -17582.072} C_VEL
LIN {X 0,Y 290.513,Z 320.555,A -85,B 0,C 180,E1 -17584.145,E2 -17584.145} C_VEL
LIN {X 0,Y 285.106,Z 312.608,A -85,B 0,C 180,E1 -17585.418,E2 -17585.418} C_VEL
LIN {X 0,Y 284.044,Z 311.03,A -85,B 0,C 180,E1 -17585.677,E2 -17585.677} C_VEL
LIN {X 0,Y 282.58,Z 309.496,A -85,B 0,C 180,E1 -17586.018,E2 -17586.018} C_VEL
LIN {X 0,Y 280.843,Z 308.527,A -85,B 0,C 180,E1 -17586.399,E2 -17586.399} C_VEL
LIN {X 0,Y 273.051,Z 305.977,A -85,B 0,C 180,E1 -17588.127,E2 -17588.127} C_VEL
LIN {X 0,Y 271.162,Z 304.015,A -85,B 0,C 180,E1 -17588.619,E2 -17588.619} C_VEL
LIN {X 0,Y 270.8,Z 303.271,A -85,B 0,C 180,E1 -17588.728,E2 -17588.728} C_VEL
LIN {X 0,Y 270.193,Z 301.132,A -85,B 0,C 180,E1 -17588.964,E2 -17588.964} C_VEL
LIN {X 0,Y 270.15,Z 301.138,A -85,B 0,C 180,E1 -17593.244,E2 -17593.244} C_VEL
LIN {X 0,Y 270.152,Z 301.133,A -85,B 0,C 180,E1 -17597.437,E2 -17597.437} C_VEL
LIN {X 0,Y 270.155,Z 301.101,A -85,B 0,C 180,E1 -17601.364,E2 -17601.364} C_VEL
LIN {X 0,Y 270.199,Z 301.089,A -85,B 0,C 180,E1 -17605.093,E2 -17605.093} C_VEL
LIN {X 0,Y 270.172,Z 301.138,A -85,B 0,C 180,E1 -17609.14,E2 -17609.14} C_VEL
LIN {X 0,Y 270.198,Z 301.13,A -85,B 0,C 180,E1 -17612.172,E2 -17612.172} C_VEL
LIN {X 0,Y 270.228,Z 301.119,A -85,B 0,C 180,E1 -17615.542,E2 -17615.542} C_VEL
LIN {X 0,Y 270.262,Z 301.128,A -85,B 0,C 180,E1 -17620.241,E2 -17620.241} C_VEL
LIN {X 0,Y 270.374,Z 301.118,A -85,B 0,C 180,E1 -17624.933,E2 -17624.933} C_VEL
LIN {X 0,Y 270.413,Z 301.1,A -85,B 0,C 180,E1 -17629.517,E2 -17629.517} C_VEL
LIN {X 0,Y 270.582,Z 301.085,A -85,B 0,C 180,E1 -17632.537,E2 -17632.537} C_VEL
LIN {X 0,Y 270.784,Z 301.062,A -85,B 0,C 180,E1 -17638.512,E2 -17638.512} C_VEL
LIN {X 0,Y 270.786,Z 301.05,A -85,B 0,C 180,E1 -17641.486,E2 -17641.486} C_VEL
LIN {X 0,Y 270.595,Z 301.058,A -85,B 0,C 180,E1 -17647.461,E2 -17647.461} C_VEL
LIN {X 0,Y 270.413,Z 301.114,A -85,B 0,C 180,E1 -17650.481,E2 -17650.481} C_VEL
LIN {X 0,Y 270.377,Z 301.116,A -85,B 0,C 180,E1 -17655.065,E2 -17655.065} C_VEL
LIN {X 0,Y 270.296,Z 301.127,A -85,B 0,C 180,E1 -17659.755,E2 -17659.755} C_VEL
LIN {X 0,Y 270.273,Z 301.132,A -85,B 0,C 180,E1 -17664.585,E2 -17664.585} C_VEL
LIN {X 0,Y 270.268,Z 301.129,A -85,B 0,C 180,E1 -17667.908,E2 -17667.908} C_VEL
LIN {X 0,Y 270.182,Z 301.141,A -85,B 0,C 180,E1 -17671.348,E2 -17671.348} C_VEL
LIN {X 0,Y 270.201,Z 301.138,A -85,B 0,C 180,E1 -17674.905,E2 -17674.905} C_VEL
LIN {X 0,Y 270.249,Z 301.142,A -85,B 0,C 180,E1 -17677.377,E2 -17677.377} C_VEL
LIN {X 0,Y 270.667,Z 302.833,A -85,B 0,C 180,E1 -17677.837,E2 -17677.837} C_VEL
LIN {X 0,Y 272.25,Z 305.265,A -85,B 0,C 180,E1 -17678.282,E2 -17678.282} C_VEL
LIN {X 0,Y 275.461,Z 310.008,A -85,B 0,C 180,E1 -17679.157,E2 -17679.157} C_VEL
LIN {X 0,Y 282.387,Z 321.125,A -85,B 0,C 180,E1 -17680.967,E2 -17680.967} C_VEL
LIN {X 0,Y 290.331,Z 334.786,A -85,B 0,C 180,E1 -17682.907,E2 -17682.907} C_VEL
LIN {X 0,Y 298.039,Z 349.47,A -85,B 0,C 180,E1 -17684.694,E2 -17684.694} C_VEL
LIN {X 0,Y 306.309,Z 367.177,A -85,B 0,C 180,E1 -17686.526,E2 -17686.526} C_VEL
LIN {X 0,Y 308.959,Z 373.342,A -85,B 0,C 180,E1 -17687.097,E2 -17687.097} C_VEL
LIN {X 0,Y 302.715,Z 510.922,A -85,B 0,C 180,E1 -17690.254,E2 -17690.254} C_VEL
LIN {X 0,Y 301.151,Z 527.74,A -85,B 0,C 180,E1 -17690.862,E2 -17690.862} C_VEL
LIN {X 0,Y 298.974,Z 543.966,A -85,B 0,C 180,E1 -17691.684,E2 -17691.684} C_VEL
LIN {X 0,Y 296.389,Z 560.183,A -85,B 0,C 180,E1 -17692.796,E2 -17692.796} C_VEL
LIN {X 0,Y 293.454,Z 575.047,A -85,B 0,C 180,E1 -17694.073,E2 -17694.073} C_VEL
LIN {X 0,Y 290.35,Z 589.447,A -85,B 0,C 180,E1 -17695.626,E2 -17695.626} C_VEL
LIN {X 0,Y 286.97,Z 603.012,A -85,B 0,C 180,E1 -17697.399,E2 -17697.399} C_VEL
LIN {X 0,Y 283.678,Z 616.087,A -85,B 0,C 180,E1 -17699.478,E2 -17699.478} C_VEL
LIN {X 0,Y 280.59,Z 627.312,A -85,B 0,C 180,E1 -17701.582,E2 -17701.582} C_VEL
LIN {X 0,Y 277.513,Z 638.467,A -85,B 0,C 180,E1 -17704.097,E2 -17704.097} C_VEL
LIN {X 0,Y 274.903,Z 647.97,A -85,B 0,C 180,E1 -17706.656,E2 -17706.656} C_VEL
LIN {X 0,Y 272.567,Z 657.195,A -85,B 0,C 180,E1 -17709.63,E2 -17709.63} C_VEL
LIN {X 0,Y 270.684,Z 664.902,A -85,B 0,C 180,E1 -17712.628,E2 -17712.628} C_VEL
LIN {X 0,Y 269.481,Z 671.175,A -85,B 0,C 180,E1 -17715.655,E2 -17715.655} C_VEL
LIN {X 0,Y 268.621,Z 676.254,A -85,B 0,C 180,E1 -17718.684,E2 -17718.684} C_VEL
LIN {X 0,Y 268.216,Z 681.02,A -85,B 0,C 180,E1 -17722.472,E2 -17722.472} C_VEL
LIN {X 0,Y 268.153,Z 683.627,A -85,B 0,C 180,E1 -17725.491,E2 -17725.491} C_VEL
LIN {X 0,Y 268.188,Z 685.204,A -85,B 0,C 180,E1 -17728.499,E2 -17728.499} C_VEL
LIN {X 0,Y 268.182,Z 685.804,A -85,B 0,C 180,E1 -17731.502,E2 -17731.502} C_VEL
LIN {X 0,Y 268.127,Z 685.217,A -85,B 0,C 180,E1 -17735.112,E2 -17735.112} C_VEL
LIN {X 0,Y 268.184,Z 684.079,A -85,B 0,C 180,E1 -17737.529,E2 -17737.529} C_VEL
LIN {X 0,Y 268.559,Z 681.773,A -85,B 0,C 180,E1 -17740.556,E2 -17740.556} C_VEL
LIN {X 0,Y 269.425,Z 678.482,A -85,B 0,C 180,E1 -17743.578,E2 -17743.578} C_VEL
LIN {X 0,Y 270.708,Z 674.149,A -85,B 0,C 180,E1 -17746.594,E2 -17746.594} C_VEL
LIN {X 0,Y 272.632,Z 668.755,A -85,B 0,C 180,E1 -17749.58,E2 -17749.58} C_VEL
LIN {X 0,Y 275.155,Z 662.12,A -85,B 0,C 180,E1 -17752.528,E2 -17752.528} C_VEL
LIN {X 0,Y 278.301,Z 654.227,A -85,B 0,C 180,E1 -17755.424,E2 -17755.424} C_VEL
LIN {X 0,Y 282.154,Z 644.845,A -85,B 0,C 180,E1 -17758.246,E2 -17758.246} C_VEL
LIN {X 0,Y 286.627,Z 633.658,A -85,B 0,C 180,E1 -17760.992,E2 -17760.992} C_VEL
LIN {X 0,Y 291.102,Z 622.104,A -85,B 0,C 180,E1 -17763.316,E2 -17763.316} C_VEL
LIN {X 0,Y 295.34,Z 610.61,A -85,B 0,C 180,E1 -17765.244,E2 -17765.244} C_VEL
LIN {X 0,Y 299.716,Z 597.635,A -85,B 0,C 180,E1 -17767.069,E2 -17767.069} C_VEL
LIN {X 0,Y 304.417,Z 582.483,A -85,B 0,C 180,E1 -17768.773,E2 -17768.773} C_VEL
LIN {X 0,Y 308.32,Z 567.959,A -85,B 0,C 180,E1 -17770.087,E2 -17770.087} C_VEL
LIN {X 0,Y 311.877,Z 552.208,A -85,B 0,C 180,E1 -17771.234,E2 -17771.234} C_VEL
LIN {X 0,Y 314.994,Z 535.678,A -85,B 0,C 180,E1 -17772.141,E2 -17772.141} C_VEL
LIN {X 0,Y 317.302,Z 519.526,A -85,B 0,C 180,E1 -17772.793,E2 -17772.793} C_VEL
LIN {X 0,Y 318.872,Z 502.467,A -85,B 0,C 180,E1 -17773.259,E2 -17773.259} C_VEL
LIN {X 0,Y 325.567,Z 383.583,A -85,B 0,C 180,E1 -17775.901,E2 -17775.901} C_VEL
LIN {X 0,Y 318.882,Z 370.285,A -85,B 0,C 180,E1 -17777.87,E2 -17777.87} C_VEL
LIN {X 0,Y 311.7,Z 357.544,A -85,B 0,C 180,E1 -17780.147,E2 -17780.147} C_VEL
LIN {X 0,Y 304.863,Z 346.627,A -85,B 0,C 180,E1 -17782.502,E2 -17782.502} C_VEL
LIN {X 0,Y 298.531,Z 337.01,A -85,B 0,C 180,E1 -17784.931,E2 -17784.931} C_VEL
LIN {X 0,Y 294.211,Z 330.908,A -85,B 0,C 180,E1 -17786.741,E2 -17786.741} C_VEL
LIN {X 0,Y 290.206,Z 325.501,A -85,B 0,C 180,E1 -17788.566,E2 -17788.566} C_VEL
LIN {X 0,Y 285.57,Z 319.415,A -85,B 0,C 180,E1 -17790.919,E2 -17790.919} C_VEL
LIN {X 0,Y 284.181,Z 317.776,A -85,B 0,C 180,E1 -17791.673,E2 -17791.673} C_VEL
LIN {X 0,Y 281.722,Z 315.137,A -85,B 0,C 180,E1 -17793.069,E2 -17793.069} C_VEL
LIN {X 0,Y 280.615,Z 312.951,A -85,B 0,C 180,E1 -17793.806,E2 -17793.806} C_VEL
LIN {X 0,Y 277.799,Z 311.059,A -85,B 0,C 180,E1 -17795.566,E2 -17795.566} C_VEL
LIN {X 0,Y 276.094,Z 308.443,A -85,B 0,C 180,E1 -17796.862,E2 -17796.862} C_VEL
LIN {X 0,Y 275.592,Z 307.121,A -85,B 0,C 180,E1 -17797.313,E2 -17797.313} C_VEL
LIN {X 0,Y 272.878,Z 305.773,A -85,B 0,C 180,E1 -17799.424,E2 -17799.424} C_VEL
LIN {X 0,Y 270.935,Z 303.285,A -85,B 0,C 180,E1 -17801.375,E2 -17801.375} C_VEL
LIN {X 0,Y 270.339,Z 301.256,A -85,B 0,C 180,E1 -17802.215,E2 -17802.215} C_VEL
LIN {X 0,Y 270.404,Z 301.09,A -85,B 0,C 180,E1 -17804.936,E2 -17804.936} C_VEL
LIN {X 0,Y 270.408,Z 301.072,A -85,B 0,C 180,E1 -17809.518,E2 -17809.518} C_VEL
LIN {X 0,Y 270.564,Z 301.097,A -85,B 0,C 180,E1 -17812.538,E2 -17812.538} C_VEL
LIN {X 0,Y 270.781,Z 301.066,A -85,B 0,C 180,E1 -17818.514,E2 -17818.514} C_VEL
LIN {X 0,Y 270.778,Z 301.028,A -85,B 0,C 180,E1 -17821.488,E2 -17821.488} C_VEL
LIN {X 0,Y 270.471,Z 301.219,A -85,B 0,C 180,E1 -17825.359,E2 -17825.359} C_VEL
LIN {X 0,Y 271.28,Z 303.488,A -85,B 0,C 180,E1 -17826.415,E2 -17826.415} C_VEL
LIN {X 0,Y 273.466,Z 305.982,A -85,B 0,C 180,E1 -17828.499,E2 -17828.499} C_VEL
LIN {X 0,Y 275.84,Z 307.358,A -85,B 0,C 180,E1 -17830.321,E2 -17830.321} C_VEL
LIN {X 0,Y 277.182,Z 310.158,A -85,B 0,C 180,E1 -17831.426,E2 -17831.426} C_VEL
LIN {X 0,Y 279.664,Z 312.381,A -85,B 0,C 180,E1 -17833.073,E2 -17833.073} C_VEL
LIN {X 0,Y 280.8,Z 313.196,A -85,B 0,C 180,E1 -17833.756,E2 -17833.756} C_VEL
LIN {X 0,Y 282.859,Z 316.546,A -85,B 0,C 180,E1 -17835.049,E2 -17835.049} C_VEL
LIN {X 0,Y 285.491,Z 318.889,A -85,B 0,C 180,E1 -17836.458,E2 -17836.458} C_VEL
LIN {X 0,Y 287.851,Z 322.237,A -85,B 0,C 180,E1 -17837.709,E2 -17837.709} C_VEL
LIN {X 0,Y 289.813,Z 324.19,A -85,B 0,C 180,E1 -17838.645,E2 -17838.645} C_VEL
LIN {X 0,Y 292.486,Z 327.793,A -85,B 0,C 180,E1 -17839.899,E2 -17839.899} C_VEL
LIN {X 0,Y 294.091,Z 329.642,A -85,B 0,C 180,E1 -17840.596,E2 -17840.596} C_VEL
LIN {X 0,Y 298.368,Z 335.133,A -85,B 0,C 180,E1 -17842.37,E2 -17842.37} C_VEL
LIN {X 0,Y 302.784,Z 341.036,A -85,B 0,C 180,E1 -17844.068,E2 -17844.068} C_VEL
LIN {X 0,Y 309.853,Z 350.763,A -85,B 0,C 180,E1 -17846.531,E2 -17846.531} C_VEL
LIN {X 0,Y 317.866,Z 362.934,A -85,B 0,C 180,E1 -17849.061,E2 -17849.061} C_VEL
LIN {X 0,Y 323.833,Z 373.002,A -85,B 0,C 180,E1 -17850.801,E2 -17850.801} C_VEL
LIN {X 0,Y 325.905,Z 377.104,A -85,B 0,C 180,E1 -17851.395,E2 -17851.395} C_VEL
LIN {X 0,Y 318.852,Z 497.811,A -85,B 0,C 180,E1 -17854.077,E2 -17854.077} C_VEL
LIN {X 0,Y 317.047,Z 513.771,A -85,B 0,C 180,E1 -17854.618,E2 -17854.618} C_VEL
LIN {X 0,Y 314.587,Z 530.227,A -85,B 0,C 180,E1 -17855.428,E2 -17855.428} C_VEL
LIN {X 0,Y 311.659,Z 545.485,A -85,B 0,C 180,E1 -17856.412,E2 -17856.412} C_VEL
LIN {X 0,Y 308.29,Z 559.959,A -85,B 0,C 180,E1 -17857.583,E2 -17857.583} C_VEL
LIN {X 0,Y 304.302,Z 574.496,A -85,B 0,C 180,E1 -17859.051,E2 -17859.051} C_VEL
LIN {X 0,Y 300.103,Z 588.023,A -85,B 0,C 180,E1 -17860.722,E2 -17860.722} C_VEL
LIN {X 0,Y 295.47,Z 601.464,A -85,B 0,C 180,E1 -17862.744,E2 -17862.744} C_VEL
LIN {X 0,Y 291.373,Z 612.498,A -85,B 0,C 180,E1 -17864.738,E2 -17864.738} C_VEL
LIN {X 0,Y 286.893,Z 623.669,A -85,B 0,C 180,E1 -17867.182,E2 -17867.182} C_VEL
LIN {X 0,Y 282.828,Z 633.38,A -85,B 0,C 180,E1 -17869.753,E2 -17869.753} C_VEL
LIN {X 0,Y 279.315,Z 641.696,A -85,B 0,C 180,E1 -17872.398,E2 -17872.398} C_VEL
LIN {X 0,Y 276.358,Z 648.685,A -85,B 0,C 180,E1 -17875.096,E2 -17875.096} C_VEL
LIN {X 0,Y 273.366,Z 655.715,A -85,B 0,C 180,E1 -17878.45,E2 -17878.45} C_VEL
LIN {X 0,Y 271.209,Z 661.129,A -85,B 0,C 180,E1 -17881.773,E2 -17881.773} C_VEL
LIN {X 0,Y 269.578,Z 665.466,A -85,B 0,C 180,E1 -17885.346,E2 -17885.346} C_VEL
LIN {X 0,Y 268.673,Z 668.094,A -85,B 0,C 180,E1 -17888.517,E2 -17888.517} C_VEL
LIN {X 0,Y 268.152,Z 669.663,A -85,B 0,C 180,E1 -17891.669,E2 -17891.669} C_VEL
LIN {X 0,Y 267.958,Z 670.236,A -85,B 0,C 180,E1 -17894.794,E2 -17894.794} C_VEL
LIN {X 0,Y 267.947,Z 669.766,A -85,B 0,C 180,E1 -17897.887,E2 -17897.887} C_VEL
LIN {X 0,Y 268.015,Z 668.383,A -85,B 0,C 180,E1 -17900.948,E2 -17900.948} C_VEL
LIN {X 0,Y 268.476,Z 665.792,A -85,B 0,C 180,E1 -17904.131,E2 -17904.131} C_VEL
LIN {X 0,Y 269.017,Z 661.512,A -85,B 0,C 180,E1 -17907.754,E2 -17907.754} C_VEL
LIN {X 0,Y 269.838,Z 656.837,A -85,B 0,C 180,E1 -17910.746,E2 -17910.746} C_VEL
LIN {X 0,Y 271.621,Z 649.313,A -85,B 0,C 180,E1 -17914.452,E2 -17914.452} C_VEL
LIN {X 0,Y 273.834,Z 640.828,A -85,B 0,C 180,E1 -17917.744,E2 -17917.744} C_VEL
LIN {X 0,Y 276.518,Z 631.67,A -85,B 0,C 180,E1 -17920.618,E2 -17920.618} C_VEL
LIN {X 0,Y 279.207,Z 622.287,A -85,B 0,C 180,E1 -17923.093,E2 -17923.093} C_VEL
LIN {X 0,Y 282.25,Z 611.389,A -85,B 0,C 180,E1 -17925.526,E2 -17925.526} C_VEL
LIN {X 0,Y 285.624,Z 598.529,A -85,B 0,C 180,E1 -17927.913,E2 -17927.913} C_VEL
LIN {X 0,Y 288.856,Z 585.43,A -85,B 0,C 180,E1 -17929.915,E2 -17929.915} C_VEL
LIN {X 0,Y 292.218,Z 571.173,A -85,B 0,C 180,E1 -17931.702,E2 -17931.702} C_VEL
LIN {X 0,Y 295.089,Z 557.285,A -85,B 0,C 180,E1 -17933.139,E2 -17933.139} C_VEL
LIN {X 0,Y 297.597,Z 542.46,A -85,B 0,C 180,E1 -17934.411,E2 -17934.411} C_VEL
LIN {X 0,Y 299.913,Z 527.14,A -85,B 0,C 180,E1 -17935.412,E2 -17935.412} C_VEL
LIN {X 0,Y 301.773,Z 510.995,A -85,B 0,C 180,E1 -17936.216,E2 -17936.216} C_VEL
LIN {X 0,Y 303.185,Z 494.505,A -85,B 0,C 180,E1 -17936.78,E2 -17936.78} C_VEL
LIN {X 0,Y 309.106,Z 366.323,A -85,B 0,C 180,E1 -17939.703,E2 -17939.703} C_VEL
LIN {X 0,Y 304.637,Z 356.539,A -85,B 0,C 180,E1 -17940.66,E2 -17940.66} C_VEL
LIN {X 0,Y 295.937,Z 340.949,A -85,B 0,C 180,E1 -17942.539,E2 -17942.539} C_VEL
LIN {X 0,Y 286.796,Z 326.099,A -85,B 0,C 180,E1 -17944.639,E2 -17944.639} C_VEL
LIN {X 0,Y 279.088,Z 314.616,A -85,B 0,C 180,E1 -17946.536,E2 -17946.536} C_VEL
LIN {X 0,Y 275.679,Z 309.925,A -85,B 0,C 180,E1 -17947.415,E2 -17947.415} C_VEL
LIN {X 0,Y 273.58,Z 306.736,A -85,B 0,C 180,E1 -17947.983,E2 -17947.983} C_VEL
LIN {X 0,Y 272.635,Z 305.629,A -85,B 0,C 180,E1 -17948.231,E2 -17948.231} C_VEL
LIN {X 0,Y 270.8,Z 303.271,A -85,B 0,C 180,E1 -17948.728,E2 -17948.728} C_VEL
LIN {X 0,Y 269.814,Z 301.888,A -85,B 0,C 180,E1 -17949.105,E2 -17949.105} C_VEL
LIN {X 0,Y 268.04,Z 301.41,A -85,B 0,C 180,E1 -17949.948,E2 -17949.948} C_VEL
LIN {X 0,Y 265.539,Z 301.708,A -85,B 0,C 180,E1 -17951.542,E2 -17951.542} C_VEL
LIN {X 0,Y 263.713,Z 302.145,A -85,B 0,C 180,E1 -17953.389,E2 -17953.389} C_VEL
LIN {X 0,Y 263.041,Z 302.017,A -85,B 0,C 180,E1 -17955.286,E2 -17955.286} C_VEL
LIN {X 0,Y 263.075,Z 302.026,A -85,B 0,C 180,E1 -17958.418,E2 -17958.418} C_VEL
LIN {X 0,Y 263.106,Z 301.965,A -85,B 0,C 180,E1 -17962.093,E2 -17962.093} C_VEL
LIN {X 0,Y 263.153,Z 301.981,A -85,B 0,C 180,E1 -17965.885,E2 -17965.885} C_VEL
LIN {X 0,Y 263.111,Z 302.012,A -85,B 0,C 180,E1 -17969.501,E2 -17969.501} C_VEL
LIN {X 0,Y 263.13,Z 302.019,A -85,B 0,C 180,E1 -17972.995,E2 -17972.995} C_VEL
LIN {X 0,Y 263.145,Z 301.998,A -85,B 0,C 180,E1 -17976.382,E2 -17976.382} C_VEL
LIN {X 0,Y 263.239,Z 302.006,A -85,B 0,C 180,E1 -17979.691,E2 -17979.691} C_VEL
LIN {X 0,Y 263.316,Z 301.997,A -85,B 0,C 180,E1 -17984.519,E2 -17984.519} C_VEL
LIN {X 0,Y 263.355,Z 301.976,A -85,B 0,C 180,E1 -17989.233,E2 -17989.233} C_VEL
LIN {X 0,Y 263.542,Z 301.965,A -85,B 0,C 180,E1 -17992.337,E2 -17992.337} C_VEL
LIN {X 0,Y 263.748,Z 301.938,A -85,B 0,C 180,E1 -17998.472,E2 -17998.472} C_VEL
LIN {X 0,Y 263.75,Z 301.926,A -85,B 0,C 180,E1 -18001.526,E2 -18001.526} C_VEL
LIN {X 0,Y 263.555,Z 301.935,A -85,B 0,C 180,E1 -18007.661,E2 -18007.661} C_VEL
LIN {X 0,Y 263.355,Z 301.994,A -85,B 0,C 180,E1 -18010.766,E2 -18010.766} C_VEL
LIN {X 0,Y 263.323,Z 301.992,A -85,B 0,C 180,E1 -18015.479,E2 -18015.479} C_VEL
LIN {X 0,Y 263.261,Z 302.007,A -85,B 0,C 180,E1 -18020.306,E2 -18020.306} C_VEL
LIN {X 0,Y 263.207,Z 302.009,A -85,B 0,C 180,E1 -18025.291,E2 -18025.291} C_VEL
LIN {X 0,Y 263.174,Z 302.014,A -85,B 0,C 180,E1 -18028.729,E2 -18028.729} C_VEL
LIN {X 0,Y 263.131,Z 302.023,A -85,B 0,C 180,E1 -18032.288,E2 -18032.288} C_VEL
LIN {X 0,Y 263.166,Z 302.007,A -85,B 0,C 180,E1 -18035.98,E2 -18035.98} C_VEL
LIN {X 0,Y 264.327,Z 305.078,A -85,B 0,C 180,E1 -18036.447,E2 -18036.447} C_VEL
LIN {X 0,Y 266.596,Z 307.479,A -85,B 0,C 180,E1 -18037.083,E2 -18037.083} C_VEL
LIN {X 0,Y 268.791,Z 310.888,A -85,B 0,C 180,E1 -18037.723,E2 -18037.723} C_VEL
LIN {X 0,Y 271.589,Z 315.148,A -85,B 0,C 180,E1 -18038.511,E2 -18038.511} C_VEL
LIN {X 0,Y 278.384,Z 326.129,A -85,B 0,C 180,E1 -18040.349,E2 -18040.349} C_VEL
LIN {X 0,Y 286.268,Z 339.911,A -85,B 0,C 180,E1 -18042.345,E2 -18042.345} C_VEL
LIN {X 0,Y 293.817,Z 354.587,A -85,B 0,C 180,E1 -18044.153,E2 -18044.153} C_VEL
LIN {X 0,Y 301.893,Z 372.142,A -85,B 0,C 180,E1 -18046.005,E2 -18046.005} C_VEL
LIN {X 0,Y 303.248,Z 375.254,A -85,B 0,C 180,E1 -18046.306,E2 -18046.306} C_VEL
LIN {X 0,Y 296.908,Z 511.195,A -85,B 0,C 180,E1 -18049.477,E2 -18049.477} C_VEL
LIN {X 0,Y 295.222,Z 528.407,A -85,B 0,C 180,E1 -18050.114,E2 -18050.114} C_VEL
LIN {X 0,Y 292.947,Z 544.719,A -85,B 0,C 180,E1 -18050.968,E2 -18050.968} C_VEL
LIN {X 0,Y 290.286,Z 560.71,A -85,B 0,C 180,E1 -18052.096,E2 -18052.096} C_VEL
LIN {X 0,Y 287.274,Z 575.427,A -85,B 0,C 180,E1 -18053.393,E2 -18053.393} C_VEL
LIN {X 0,Y 283.909,Z 590.504,A -85,B 0,C 180,E1 -18055.063,E2 -18055.063} C_VEL
LIN {X 0,Y 280.318,Z 604.444,A -85,B 0,C 180,E1 -18056.955,E2 -18056.955} C_VEL
LIN {X 0,Y 276.889,Z 617.236,A -85,B 0,C 180,E1 -18059.07,E2 -18059.07} C_VEL
LIN {X 0,Y 273.735,Z 628.238,A -85,B 0,C 180,E1 -18061.224,E2 -18061.224} C_VEL
LIN {X 0,Y 270.583,Z 639.28,A -85,B 0,C 180,E1 -18063.797,E2 -18063.797} C_VEL
LIN {X 0,Y 267.557,Z 649.987,A -85,B 0,C 180,E1 -18066.83,E2 -18066.83} C_VEL
LIN {X 0,Y 265.233,Z 658.727,A -85,B 0,C 180,E1 -18069.851,E2 -18069.851} C_VEL
LIN {X 0,Y 263.43,Z 666.093,A -85,B 0,C 180,E1 -18072.935,E2 -18072.935} C_VEL
LIN {X 0,Y 262.22,Z 672.182,A -85,B 0,C 180,E1 -18076.042,E2 -18076.042} C_VEL
LIN {X 0,Y 261.424,Z 676.97,A -85,B 0,C 180,E1 -18079.153,E2 -18079.153} C_VEL
LIN {X 0,Y 261.123,Z 680.701,A -85,B 0,C 180,E1 -18082.266,E2 -18082.266} C_VEL
LIN {X 0,Y 261.128,Z 682.883,A -85,B 0,C 180,E1 -18084.751,E2 -18084.751} C_VEL
LIN {X 0,Y 261.115,Z 684.962,A -85,B 0,C 180,E1 -18088.458,E2 -18088.458} C_VEL
LIN {X 0,Y 261.109,Z 685.584,A -85,B 0,C 180,E1 -18091.543,E2 -18091.543} C_VEL
LIN {X 0,Y 261.05,Z 685.107,A -85,B 0,C 180,E1 -18095.06,E2 -18095.06} C_VEL
LIN {X 0,Y 261.103,Z 683.931,A -85,B 0,C 180,E1 -18097.735,E2 -18097.735} C_VEL
LIN {X 0,Y 261.505,Z 681.676,A -85,B 0,C 180,E1 -18100.844,E2 -18100.844} C_VEL
LIN {X 0,Y 262.437,Z 678.412,A -85,B 0,C 180,E1 -18103.947,E2 -18103.947} C_VEL
LIN {X 0,Y 263.812,Z 674.135,A -85,B 0,C 180,E1 -18107.04,E2 -18107.04} C_VEL
LIN {X 0,Y 265.866,Z 668.769,A -85,B 0,C 180,E1 -18110.099,E2 -18110.099} C_VEL
LIN {X 0,Y 268.501,Z 662.195,A -85,B 0,C 180,E1 -18113.118,E2 -18113.118} C_VEL
LIN {X 0,Y 271.831,Z 654.374,A -85,B 0,C 180,E1 -18116.074,E2 -18116.074} C_VEL
LIN {X 0,Y 275.862,Z 645.038,A -85,B 0,C 180,E1 -18118.951,E2 -18118.951} C_VEL
LIN {X 0,Y 279.827,Z 635.584,A -85,B 0,C 180,E1 -18121.36,E2 -18121.36} C_VEL
LIN {X 0,Y 284.507,Z 624.243,A -85,B 0,C 180,E1 -18123.766,E2 -18123.766} C_VEL
LIN {X 0,Y 288.043,Z 615.06,A -85,B 0,C 180,E1 -18125.414,E2 -18125.414} C_VEL
LIN {X 0,Y 292.788,Z 602.136,A -85,B 0,C 180,E1 -18127.362,E2 -18127.362} C_VEL
LIN {X 0,Y 296.821,Z 590.173,A -85,B 0,C 180,E1 -18128.863,E2 -18128.863} C_VEL
LIN {X 0,Y 301.16,Z 575.599,A -85,B 0,C 180,E1 -18130.36,E2 -18130.36} C_VEL
LIN {X 0,Y 304.834,Z 561.615,A -85,B 0,C 180,E1 -18131.517,E2 -18131.517} C_VEL
LIN {X 0,Y 308.103,Z 546.771,A -85,B 0,C 180,E1 -18132.514,E2 -18132.514} C_VEL
LIN {X 0,Y 311.023,Z 530.518,A -85,B 0,C 180,E1 -18133.323,E2 -18133.323} C_VEL
LIN {X 0,Y 313.008,Z 515.638,A -85,B 0,C 180,E1 -18133.86,E2 -18133.86} C_VEL
LIN {X 0,Y 314.518,Z 495.517,A -85,B 0,C 180,E1 -18134.387,E2 -18134.387} C_VEL
LIN {X 0,Y 320.944,Z 386.51,A -85,B 0,C 180,E1 -18136.81,E2 -18136.81} C_VEL
LIN {X 0,Y 314.878,Z 374.36,A -85,B 0,C 180,E1 -18138.682,E2 -18138.682} C_VEL
LIN {X 0,Y 308.39,Z 362.659,A -85,B 0,C 180,E1 -18140.827,E2 -18140.827} C_VEL
LIN {X 0,Y 302.114,Z 352.426,A -85,B 0,C 180,E1 -18143.072,E2 -18143.072} C_VEL
LIN {X 0,Y 295.639,Z 342.418,A -85,B 0,C 180,E1 -18145.653,E2 -18145.653} C_VEL
LIN {X 0,Y 291.772,Z 336.895,A -85,B 0,C 180,E1 -18147.335,E2 -18147.335} C_VEL
LIN {X 0,Y 288.255,Z 331.977,A -85,B 0,C 180,E1 -18149,E2 -18149} C_VEL
LIN {X 0,Y 282.901,Z 324.751,A -85,B 0,C 180,E1 -18151.836,E2 -18151.836} C_VEL
LIN {X 0,Y 280.163,Z 321.936,A -85,B 0,C 180,E1 -18153.41,E2 -18153.41} C_VEL
LIN {X 0,Y 278.79,Z 319.628,A -85,B 0,C 180,E1 -18154.325,E2 -18154.325} C_VEL
LIN {X 0,Y 276.029,Z 317.458,A -85,B 0,C 180,E1 -18156.143,E2 -18156.143} C_VEL
LIN {X 0,Y 274.245,Z 314.362,A -85,B 0,C 180,E1 -18157.593,E2 -18157.593} C_VEL
LIN {X 0,Y 274.038,Z 313.967,A -85,B 0,C 180,E1 -18157.774,E2 -18157.774} C_VEL
LIN {X 0,Y 271.287,Z 312.31,A -85,B 0,C 180,E1 -18160.035,E2 -18160.035} C_VEL
LIN {X 0,Y 269.478,Z 309.626,A -85,B 0,C 180,E1 -18162.009,E2 -18162.009} C_VEL
LIN {X 0,Y 268.998,Z 308.063,A -85,B 0,C 180,E1 -18162.712,E2 -18162.712} C_VEL
LIN {X 0,Y 265.409,Z 306.138,A -85,B 0,C 180,E1 -18168.206,E2 -18168.206} C_VEL
LIN {X 0,Y 264.369,Z 304.585,A -85,B 0,C 180,E1 -18172.362,E2 -18172.362} C_VEL
LIN {X 0,Y 264.312,Z 304.649,A -85,B 0,C 180,E1 -18174.661,E2 -18174.661} C_VEL
LIN {X 0,Y 265.457,Z 305.76,A -85,B 0,C 180,E1 -18179.242,E2 -18179.242} C_VEL
LIN {X 0,Y 268.791,Z 308,A -85,B 0,C 180,E1 -18184.5,E2 -18184.5} C_VEL
LIN {X 0,Y 269.26,Z 308.398,A -85,B 0,C 180,E1 -18185.055,E2 -18185.055} C_VEL
LIN {X 0,Y 270.448,Z 310.97,A -85,B 0,C 180,E1 -18186.529,E2 -18186.529} C_VEL
LIN {X 0,Y 273.026,Z 313.375,A -85,B 0,C 180,E1 -18188.886,E2 -18188.886} C_VEL
LIN {X 0,Y 274.347,Z 314.226,A -85,B 0,C 180,E1 -18189.912,E2 -18189.912} C_VEL
LIN {X 0,Y 275.88,Z 317.105,A -85,B 0,C 180,E1 -18191.178,E2 -18191.178} C_VEL
LIN {X 0,Y 278.441,Z 319.325,A -85,B 0,C 180,E1 -18192.899,E2 -18192.899} C_VEL
LIN {X 0,Y 279.251,Z 320.152,A -85,B 0,C 180,E1 -18193.416,E2 -18193.416} C_VEL
LIN {X 0,Y 281.488,Z 323.481,A -85,B 0,C 180,E1 -18194.828,E2 -18194.828} C_VEL
LIN {X 0,Y 283.783,Z 325.712,A -85,B 0,C 180,E1 -18196.092,E2 -18196.092} C_VEL
LIN {X 0,Y 286.47,Z 329.237,A -85,B 0,C 180,E1 -18197.526,E2 -18197.526} C_VEL
LIN {X 0,Y 287.785,Z 330.641,A -85,B 0,C 180,E1 -18198.172,E2 -18198.172} C_VEL
LIN {X 0,Y 290.697,Z 334.488,A -85,B 0,C 180,E1 -18199.571,E2 -18199.571} C_VEL
LIN {X 0,Y 292.176,Z 336.375,A -85,B 0,C 180,E1 -18200.236,E2 -18200.236} C_VEL
LIN {X 0,Y 295.898,Z 341.141,A -85,B 0,C 180,E1 -18201.82,E2 -18201.82} C_VEL
LIN {X 0,Y 301.849,Z 349.214,A -85,B 0,C 180,E1 -18204.148,E2 -18204.148} C_VEL
LIN {X 0,Y 309.471,Z 360.26,A -85,B 0,C 180,E1 -18206.815,E2 -18206.815} C_VEL
LIN {X 0,Y 316.645,Z 371.669,A -85,B 0,C 180,E1 -18209.093,E2 -18209.093} C_VEL
LIN {X 0,Y 320.821,Z 379.188,A -85,B 0,C 180,E1 -18210.347,E2 -18210.347} C_VEL
LIN {X 0,Y 321.274,Z 380.087,A -85,B 0,C 180,E1 -18210.481,E2 -18210.481} C_VEL
LIN {X 0,Y 314.144,Z 497.939,A -85,B 0,C 180,E1 -18213.117,E2 -18213.117} C_VEL
LIN {X 0,Y 312.265,Z 513.89,A -85,B 0,C 180,E1 -18213.653,E2 -18213.653} C_VEL
LIN {X 0,Y 309.744,Z 530.326,A -85,B 0,C 180,E1 -18214.466,E2 -18214.466} C_VEL
LIN {X 0,Y 306.785,Z 545.392,A -85,B 0,C 180,E1 -18215.444,E2 -18215.444} C_VEL
LIN {X 0,Y 303.249,Z 560.071,A -85,B 0,C 180,E1 -18216.635,E2 -18216.635} C_VEL
LIN {X 0,Y 299.16,Z 574.455,A -85,B 0,C 180,E1 -18218.094,E2 -18218.094} C_VEL
LIN {X 0,Y 294.845,Z 587.89,A -85,B 0,C 180,E1 -18219.761,E2 -18219.761} C_VEL
LIN {X 0,Y 290.358,Z 600.466,A -85,B 0,C 180,E1 -18221.641,E2 -18221.641} C_VEL
LIN {X 0,Y 285.838,Z 612.299,A -85,B 0,C 180,E1 -18223.792,E2 -18223.792} C_VEL
LIN {X 0,Y 281.111,Z 623.555,A -85,B 0,C 180,E1 -18226.269,E2 -18226.269} C_VEL
LIN {X 0,Y 277.042,Z 632.829,A -85,B 0,C 180,E1 -18228.733,E2 -18228.733} C_VEL
LIN {X 0,Y 273.286,Z 641.275,A -85,B 0,C 180,E1 -18231.418,E2 -18231.418} C_VEL
LIN {X 0,Y 270.005,Z 648.563,A -85,B 0,C 180,E1 -18234.266,E2 -18234.266} C_VEL
LIN {X 0,Y 267.089,Z 655.046,A -85,B 0,C 180,E1 -18237.356,E2 -18237.356} C_VEL
LIN {X 0,Y 264.791,Z 660.464,A -85,B 0,C 180,E1 -18240.593,E2 -18240.593} C_VEL
LIN {X 0,Y 262.733,Z 665.455,A -85,B 0,C 180,E1 -18244.659,E2 -18244.659} C_VEL
LIN {X 0,Y 261.713,Z 668.135,A -85,B 0,C 180,E1 -18247.916,E2 -18247.916} C_VEL
LIN {X 0,Y 261.118,Z 669.803,A -85,B 0,C 180,E1 -18251.157,E2 -18251.157} C_VEL
LIN {X 0,Y 260.868,Z 670.424,A -85,B 0,C 180,E1 -18254.371,E2 -18254.371} C_VEL
LIN {X 0,Y 260.84,Z 670.051,A -85,B 0,C 180,E1 -18257.552,E2 -18257.552} C_VEL
LIN {X 0,Y 260.887,Z 668.715,A -85,B 0,C 180,E1 -18260.698,E2 -18260.698} C_VEL
LIN {X 0,Y 261.398,Z 666.043,A -85,B 0,C 180,E1 -18264.158,E2 -18264.158} C_VEL
LIN {X 0,Y 261.889,Z 662.042,A -85,B 0,C 180,E1 -18267.693,E2 -18267.693} C_VEL
LIN {X 0,Y 262.755,Z 657.418,A -85,B 0,C 180,E1 -18270.766,E2 -18270.766} C_VEL
LIN {X 0,Y 264.145,Z 651.606,A -85,B 0,C 180,E1 -18273.814,E2 -18273.814} C_VEL
LIN {X 0,Y 265.968,Z 644.621,A -85,B 0,C 180,E1 -18276.829,E2 -18276.829} C_VEL
LIN {X 0,Y 268.438,Z 636.207,A -85,B 0,C 180,E1 -18279.798,E2 -18279.798} C_VEL
LIN {X 0,Y 271.098,Z 627.484,A -85,B 0,C 180,E1 -18282.349,E2 -18282.349} C_VEL
LIN {X 0,Y 274.115,Z 617.405,A -85,B 0,C 180,E1 -18284.856,E2 -18284.856} C_VEL
LIN {X 0,Y 277.443,Z 605.614,A -85,B 0,C 180,E1 -18287.316,E2 -18287.316} C_VEL
LIN {X 0,Y 280.947,Z 592.625,A -85,B 0,C 180,E1 -18289.547,E2 -18289.547} C_VEL
LIN {X 0,Y 284.137,Z 579.688,A -85,B 0,C 180,E1 -18291.397,E2 -18291.397} C_VEL
LIN {X 0,Y 287.335,Z 565.807,A -85,B 0,C 180,E1 -18293.038,E2 -18293.038} C_VEL
LIN {X 0,Y 290.239,Z 550.85,A -85,B 0,C 180,E1 -18294.499,E2 -18294.499} C_VEL
LIN {X 0,Y 292.652,Z 536.425,A -85,B 0,C 180,E1 -18295.611,E2 -18295.611} C_VEL
LIN {X 0,Y 295.011,Z 520.009,A -85,B 0,C 180,E1 -18296.578,E2 -18296.578} C_VEL
LIN {X 0,Y 296.686,Z 504.042,A -85,B 0,C 180,E1 -18297.272,E2 -18297.272} C_VEL
LIN {X 0,Y 297.93,Z 486.573,A -85,B 0,C 180,E1 -18297.768,E2 -18297.768} C_VEL
LIN {X 0,Y 303.468,Z 368.528,A -85,B 0,C 180,E1 -18300.478,E2 -18300.478} C_VEL
LIN {X 0,Y 299.584,Z 360.065,A -85,B 0,C 180,E1 -18301.342,E2 -18301.342} C_VEL
LIN {X 0,Y 291.032,Z 344.751,A -85,B 0,C 180,E1 -18303.257,E2 -18303.257} C_VEL
LIN {X 0,Y 282.349,Z 330.554,A -85,B 0,C 180,E1 -18305.327,E2 -18305.327} C_VEL
LIN {X 0,Y 274.819,Z 319.293,A -85,B 0,C 180,E1 -18307.252,E2 -18307.252} C_VEL
LIN {X 0,Y 271.514,Z 314.683,A -85,B 0,C 180,E1 -18308.135,E2 -18308.135} C_VEL
LIN {X 0,Y 269.125,Z 311.272,A -85,B 0,C 180,E1 -18308.799,E2 -18308.799} C_VEL
LIN {X 0,Y 266.721,Z 307.877,A -85,B 0,C 180,E1 -18309.486,E2 -18309.486} C_VEL
LIN {X 0,Y 266.119,Z 306.976,A -85,B 0,C 180,E1 -18309.663,E2 -18309.663} C_VEL
LIN {X 0,Y 263.977,Z 304.654,A -85,B 0,C 180,E1 -18310.27,E2 -18310.27} C_VEL
LIN {X 0,Y 263.109,Z 302.02,A -85,B 0,C 180,E1 -18310.599,E2 -18310.599} C_VEL
LIN {X 0,Y 263.079,Z 302.027,A -85,B 0,C 180,E1 -18313.993,E2 -18313.993} C_VEL
LIN {X 0,Y 263.041,Z 302.017,A -85,B 0,C 180,E1 -18315.286,E2 -18315.286} C_VEL
LIN {X 0,Y 262.393,Z 302.101,A -85,B 0,C 180,E1 -18316.564,E2 -18316.564} C_VEL
LIN {X 0,Y 259.531,Z 302.47,A -85,B 0,C 180,E1 -18318.646,E2 -18318.646} C_VEL
LIN {X 0,Y 257.11,Z 302.748,A -85,B 0,C 180,E1 -18320.341,E2 -18320.341} C_VEL
LIN {X 0,Y 256.105,Z 302.842,A -85,B 0,C 180,E1 -18321.655,E2 -18321.655} C_VEL
LIN {X 0,Y 256.042,Z 302.843,A -85,B 0,C 180,E1 -18322.1,E2 -18322.1} C_VEL
LIN {X 0,Y 256.106,Z 302.847,A -85,B 0,C 180,E1 -18325.412,E2 -18325.412} C_VEL
LIN {X 0,Y 256.079,Z 302.898,A -85,B 0,C 180,E1 -18328.57,E2 -18328.57} C_VEL
LIN {X 0,Y 256.087,Z 302.887,A -85,B 0,C 180,E1 -18332.189,E2 -18332.189} C_VEL
LIN {X 0,Y 256.134,Z 302.873,A -85,B 0,C 180,E1 -18335.695,E2 -18335.695} C_VEL
LIN {X 0,Y 256.148,Z 302.891,A -85,B 0,C 180,E1 -18339.102,E2 -18339.102} C_VEL
LIN {X 0,Y 256.25,Z 302.871,A -85,B 0,C 180,E1 -18344.081,E2 -18344.081} C_VEL
LIN {X 0,Y 256.291,Z 302.853,A -85,B 0,C 180,E1 -18347.327,E2 -18347.327} C_VEL
LIN {X 0,Y 256.503,Z 302.843,A -85,B 0,C 180,E1 -18352.125,E2 -18352.125} C_VEL
LIN {X 0,Y 256.486,Z 302.847,A -85,B 0,C 180,E1 -18356.858,E2 -18356.858} C_VEL
LIN {X 0,Y 256.758,Z 302.791,A -85,B 0,C 180,E1 -18359.999,E2 -18359.999} C_VEL
LIN {X 0,Y 256.497,Z 302.847,A -85,B 0,C 180,E1 -18363.141,E2 -18363.141} C_VEL
LIN {X 0,Y 256.513,Z 302.813,A -85,B 0,C 180,E1 -18367.873,E2 -18367.873} C_VEL
LIN {X 0,Y 256.289,Z 302.866,A -85,B 0,C 180,E1 -18372.672,E2 -18372.672} C_VEL
LIN {X 0,Y 256.242,Z 302.874,A -85,B 0,C 180,E1 -18376.271,E2 -18376.271} C_VEL
LIN {X 0,Y 256.166,Z 302.893,A -85,B 0,C 180,E1 -18380.894,E2 -18380.894} C_VEL
LIN {X 0,Y 256.187,Z 302.884,A -85,B 0,C 180,E1 -18385.138,E2 -18385.138} C_VEL
LIN {X 0,Y 256.109,Z 302.898,A -85,B 0,C 180,E1 -18389.599,E2 -18389.599} C_VEL
LIN {X 0,Y 256.133,Z 302.961,A -85,B 0,C 180,E1 -18394.268,E2 -18394.268} C_VEL
LIN {X 0,Y 257.051,Z 305.645,A -85,B 0,C 180,E1 -18394.629,E2 -18394.629} C_VEL
LIN {X 0,Y 258.964,Z 307.728,A -85,B 0,C 180,E1 -18395.218,E2 -18395.218} C_VEL
LIN {X 0,Y 259.745,Z 308.544,A -85,B 0,C 180,E1 -18395.452,E2 -18395.452} C_VEL
LIN {X 0,Y 261.882,Z 311.848,A -85,B 0,C 180,E1 -18396.125,E2 -18396.125} C_VEL
LIN {X 0,Y 263.289,Z 313.514,A -85,B 0,C 180,E1 -18396.536,E2 -18396.536} C_VEL
LIN {X 0,Y 267.874,Z 320.458,A -85,B 0,C 180,E1 -18397.885,E2 -18397.885} C_VEL
LIN {X 0,Y 274.13,Z 330.674,A -85,B 0,C 180,E1 -18399.637,E2 -18399.637} C_VEL
LIN {X 0,Y 281.904,Z 344.457,A -85,B 0,C 180,E1 -18401.684,E2 -18401.684} C_VEL
LIN {X 0,Y 289.152,Z 358.727,A -85,B 0,C 180,E1 -18403.486,E2 -18403.486} C_VEL
LIN {X 0,Y 297.274,Z 376.648,A -85,B 0,C 180,E1 -18405.417,E2 -18405.417} C_VEL
LIN {X 0,Y 297.626,Z 377.442,A -85,B 0,C 180,E1 -18405.498,E2 -18405.498} C_VEL
LIN {X 0,Y 291.214,Z 510.223,A -85,B 0,C 180,E1 -18408.637,E2 -18408.637} C_VEL
LIN {X 0,Y 289.612,Z 526.659,A -85,B 0,C 180,E1 -18409.237,E2 -18409.237} C_VEL
LIN {X 0,Y 287.405,Z 542.769,A -85,B 0,C 180,E1 -18410.067,E2 -18410.067} C_VEL
LIN {X 0,Y 284.786,Z 558.151,A -85,B 0,C 180,E1 -18411.116,E2 -18411.116} C_VEL
LIN {X 0,Y 282.307,Z 570.633,A -85,B 0,C 180,E1 -18412.191,E2 -18412.191} C_VEL
LIN {X 0,Y 278.896,Z 585.47,A -85,B 0,C 180,E1 -18413.742,E2 -18413.742} C_VEL
LIN {X 0,Y 275.279,Z 599.878,A -85,B 0,C 180,E1 -18415.607,E2 -18415.607} C_VEL
LIN {X 0,Y 271.926,Z 612.39,A -85,B 0,C 180,E1 -18417.569,E2 -18417.569} C_VEL
LIN {X 0,Y 268.368,Z 624.222,A -85,B 0,C 180,E1 -18419.79,E2 -18419.79} C_VEL
LIN {X 0,Y 265.047,Z 635.57,A -85,B 0,C 180,E1 -18422.353,E2 -18422.353} C_VEL
LIN {X 0,Y 262.016,Z 645.487,A -85,B 0,C 180,E1 -18425.01,E2 -18425.01} C_VEL
LIN {X 0,Y 259.307,Z 655.073,A -85,B 0,C 180,E1 -18428.12,E2 -18428.12} C_VEL
LIN {X 0,Y 257.391,Z 662.077,A -85,B 0,C 180,E1 -18430.874,E2 -18430.874} C_VEL
LIN {X 0,Y 255.774,Z 668.916,A -85,B 0,C 180,E1 -18434.09,E2 -18434.09} C_VEL
LIN {X 0,Y 254.784,Z 674.315,A -85,B 0,C 180,E1 -18437.252,E2 -18437.252} C_VEL
LIN {X 0,Y 254.177,Z 678.611,A -85,B 0,C 180,E1 -18440.451,E2 -18440.451} C_VEL
LIN {X 0,Y 254.025,Z 681.858,A -85,B 0,C 180,E1 -18443.646,E2 -18443.646} C_VEL
LIN {X 0,Y 253.984,Z 683.991,A -85,B 0,C 180,E1 -18446.828,E2 -18446.828} C_VEL
LIN {X 0,Y 254.052,Z 685.187,A -85,B 0,C 180,E1 -18450,E2 -18450} C_VEL
LIN {X 0,Y 253.936,Z 685.325,A -85,B 0,C 180,E1 -18453.173,E2 -18453.173} C_VEL
LIN {X 0,Y 253.945,Z 684.566,A -85,B 0,C 180,E1 -18456.356,E2 -18456.356} C_VEL
LIN {X 0,Y 254.215,Z 682.79,A -85,B 0,C 180,E1 -18459.548,E2 -18459.548} C_VEL
LIN {X 0,Y 254.921,Z 680.102,A -85,B 0,C 180,E1 -18462.742,E2 -18462.742} C_VEL
